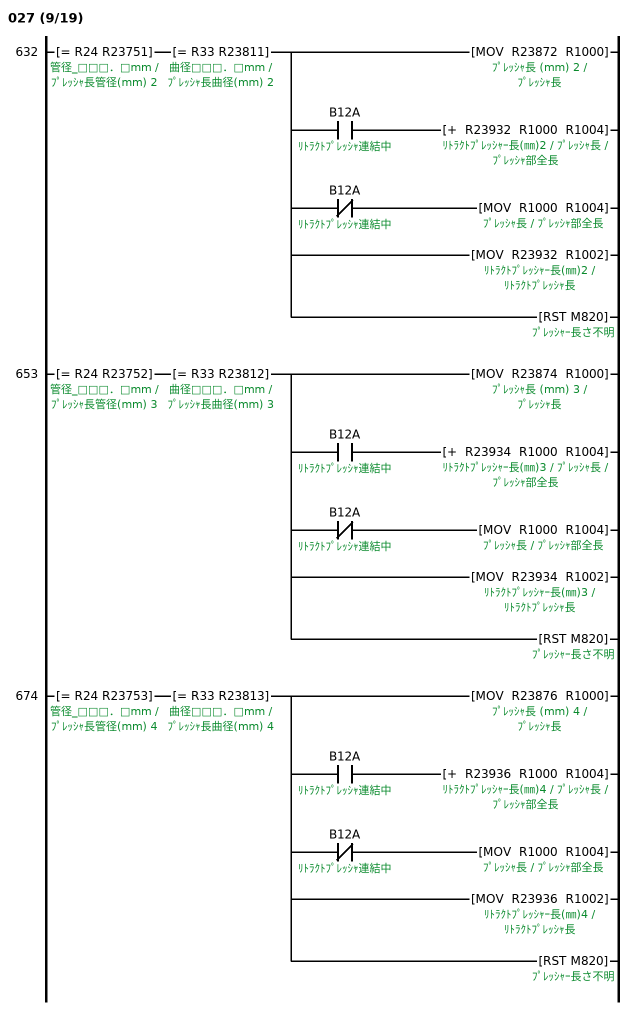
632   LD=     R24 R23751  ; 管径_□□□．□mm / ﾌﾟﾚｯｼｬ長管径(mm) 2
      AND=    R33 R23811  ; 曲径□□□．□mm / ﾌﾟﾚｯｼｬ長曲径(mm) 2
      MOV     R23872 R1000  ; ﾌﾟﾚｯｼｬ長 (mm) 2
      MPS
      AND     B12A  ; ﾘﾄﾗｸﾄﾌﾟﾚｯｼｬ連結中
      +       R23932 R1000 R1004  ; ﾘﾄﾗｸﾄﾌﾟﾚｯｼｬｰ長(㎜)2
      MRD
      ANI     B12A  ; ﾘﾄﾗｸﾄﾌﾟﾚｯｼｬ連結中
      MOV     R1000 R1004
      MPP
      MOV     R23932 R1002
      RST     M820  ; ﾌﾟﾚｯｼｬｰ長さ不明
653   LD=     R24 R23752  ; 管径_□□□．□mm / ﾌﾟﾚｯｼｬ長管径(mm) 3
      AND=    R33 R23812  ; 曲径□□□．□mm / ﾌﾟﾚｯｼｬ長曲径(mm) 3
      MOV     R23874 R1000  ; ﾌﾟﾚｯｼｬ長 (mm) 3
      MPS
      AND     B12A  ; ﾘﾄﾗｸﾄﾌﾟﾚｯｼｬ連結中
      +       R23934 R1000 R1004  ; ﾘﾄﾗｸﾄﾌﾟﾚｯｼｬｰ長(㎜)3
      MRD
      ANI     B12A  ; ﾘﾄﾗｸﾄﾌﾟﾚｯｼｬ連結中
      MOV     R1000 R1004
      MPP
      MOV     R23934 R1002
      RST     M820  ; ﾌﾟﾚｯｼｬｰ長さ不明
674   LD=     R24 R23753  ; 管径_□□□．□mm / ﾌﾟﾚｯｼｬ長管径(mm) 4
      AND=    R33 R23813  ; 曲径□□□．□mm / ﾌﾟﾚｯｼｬ長曲径(mm) 4
      MOV     R23876 R1000  ; ﾌﾟﾚｯｼｬ長 (mm) 4
      MPS
      AND     B12A  ; ﾘﾄﾗｸﾄﾌﾟﾚｯｼｬ連結中
      +       R23936 R1000 R1004  ; ﾘﾄﾗｸﾄﾌﾟﾚｯｼｬｰ長(㎜)4
      MRD
      ANI     B12A  ; ﾘﾄﾗｸﾄﾌﾟﾚｯｼｬ連結中
      MOV     R1000 R1004
      MPP
      MOV     R23936 R1002
      RST     M820  ; ﾌﾟﾚｯｼｬｰ長さ不明
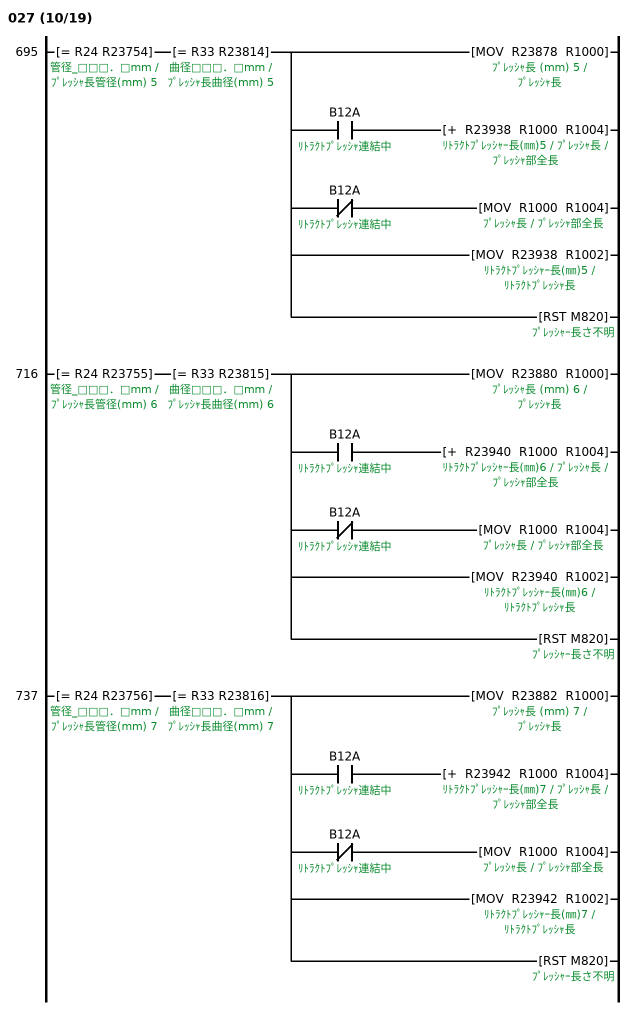
695   LD=     R24 R23754  ; 管径_□□□．□mm / ﾌﾟﾚｯｼｬ長管径(mm) 5
      AND=    R33 R23814  ; 曲径□□□．□mm / ﾌﾟﾚｯｼｬ長曲径(mm) 5
      MOV     R23878 R1000  ; ﾌﾟﾚｯｼｬ長 (mm) 5
      MPS
      AND     B12A  ; ﾘﾄﾗｸﾄﾌﾟﾚｯｼｬ連結中
      +       R23938 R1000 R1004  ; ﾘﾄﾗｸﾄﾌﾟﾚｯｼｬｰ長(㎜)5
      MRD
      ANI     B12A  ; ﾘﾄﾗｸﾄﾌﾟﾚｯｼｬ連結中
      MOV     R1000 R1004
      MPP
      MOV     R23938 R1002
      RST     M820  ; ﾌﾟﾚｯｼｬｰ長さ不明
716   LD=     R24 R23755  ; 管径_□□□．□mm / ﾌﾟﾚｯｼｬ長管径(mm) 6
      AND=    R33 R23815  ; 曲径□□□．□mm / ﾌﾟﾚｯｼｬ長曲径(mm) 6
      MOV     R23880 R1000  ; ﾌﾟﾚｯｼｬ長 (mm) 6
      MPS
      AND     B12A  ; ﾘﾄﾗｸﾄﾌﾟﾚｯｼｬ連結中
      +       R23940 R1000 R1004  ; ﾘﾄﾗｸﾄﾌﾟﾚｯｼｬｰ長(㎜)6
      MRD
      ANI     B12A  ; ﾘﾄﾗｸﾄﾌﾟﾚｯｼｬ連結中
      MOV     R1000 R1004
      MPP
      MOV     R23940 R1002
      RST     M820  ; ﾌﾟﾚｯｼｬｰ長さ不明
737   LD=     R24 R23756  ; 管径_□□□．□mm / ﾌﾟﾚｯｼｬ長管径(mm) 7
      AND=    R33 R23816  ; 曲径□□□．□mm / ﾌﾟﾚｯｼｬ長曲径(mm) 7
      MOV     R23882 R1000  ; ﾌﾟﾚｯｼｬ長 (mm) 7
      MPS
      AND     B12A  ; ﾘﾄﾗｸﾄﾌﾟﾚｯｼｬ連結中
      +       R23942 R1000 R1004  ; ﾘﾄﾗｸﾄﾌﾟﾚｯｼｬｰ長(㎜)7
      MRD
      ANI     B12A  ; ﾘﾄﾗｸﾄﾌﾟﾚｯｼｬ連結中
      MOV     R1000 R1004
      MPP
      MOV     R23942 R1002
      RST     M820  ; ﾌﾟﾚｯｼｬｰ長さ不明
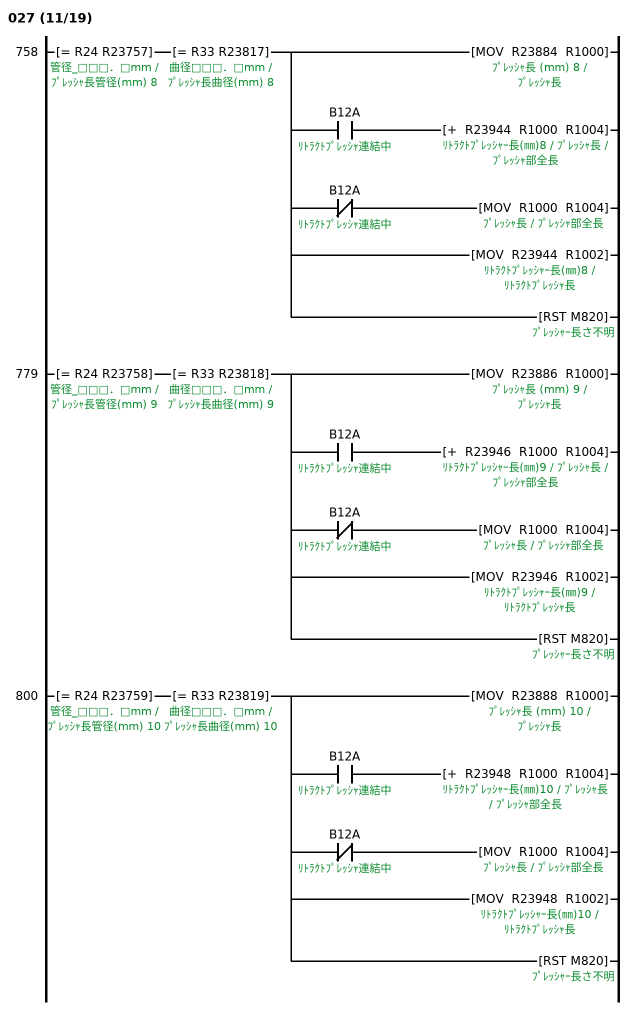
758   LD=     R24 R23757  ; 管径_□□□．□mm / ﾌﾟﾚｯｼｬ長管径(mm) 8
      AND=    R33 R23817  ; 曲径□□□．□mm / ﾌﾟﾚｯｼｬ長曲径(mm) 8
      MOV     R23884 R1000  ; ﾌﾟﾚｯｼｬ長 (mm) 8
      MPS
      AND     B12A  ; ﾘﾄﾗｸﾄﾌﾟﾚｯｼｬ連結中
      +       R23944 R1000 R1004  ; ﾘﾄﾗｸﾄﾌﾟﾚｯｼｬｰ長(㎜)8
      MRD
      ANI     B12A  ; ﾘﾄﾗｸﾄﾌﾟﾚｯｼｬ連結中
      MOV     R1000 R1004
      MPP
      MOV     R23944 R1002
      RST     M820  ; ﾌﾟﾚｯｼｬｰ長さ不明
779   LD=     R24 R23758  ; 管径_□□□．□mm / ﾌﾟﾚｯｼｬ長管径(mm) 9
      AND=    R33 R23818  ; 曲径□□□．□mm / ﾌﾟﾚｯｼｬ長曲径(mm) 9
      MOV     R23886 R1000  ; ﾌﾟﾚｯｼｬ長 (mm) 9
      MPS
      AND     B12A  ; ﾘﾄﾗｸﾄﾌﾟﾚｯｼｬ連結中
      +       R23946 R1000 R1004  ; ﾘﾄﾗｸﾄﾌﾟﾚｯｼｬｰ長(㎜)9
      MRD
      ANI     B12A  ; ﾘﾄﾗｸﾄﾌﾟﾚｯｼｬ連結中
      MOV     R1000 R1004
      MPP
      MOV     R23946 R1002
      RST     M820  ; ﾌﾟﾚｯｼｬｰ長さ不明
800   LD=     R24 R23759  ; 管径_□□□．□mm / ﾌﾟﾚｯｼｬ長管径(mm) 10
      AND=    R33 R23819  ; 曲径□□□．□mm / ﾌﾟﾚｯｼｬ長曲径(mm) 10
      MOV     R23888 R1000  ; ﾌﾟﾚｯｼｬ長 (mm) 10
      MPS
      AND     B12A  ; ﾘﾄﾗｸﾄﾌﾟﾚｯｼｬ連結中
      +       R23948 R1000 R1004  ; ﾘﾄﾗｸﾄﾌﾟﾚｯｼｬｰ長(㎜)10
      MRD
      ANI     B12A  ; ﾘﾄﾗｸﾄﾌﾟﾚｯｼｬ連結中
      MOV     R1000 R1004
      MPP
      MOV     R23948 R1002
      RST     M820  ; ﾌﾟﾚｯｼｬｰ長さ不明
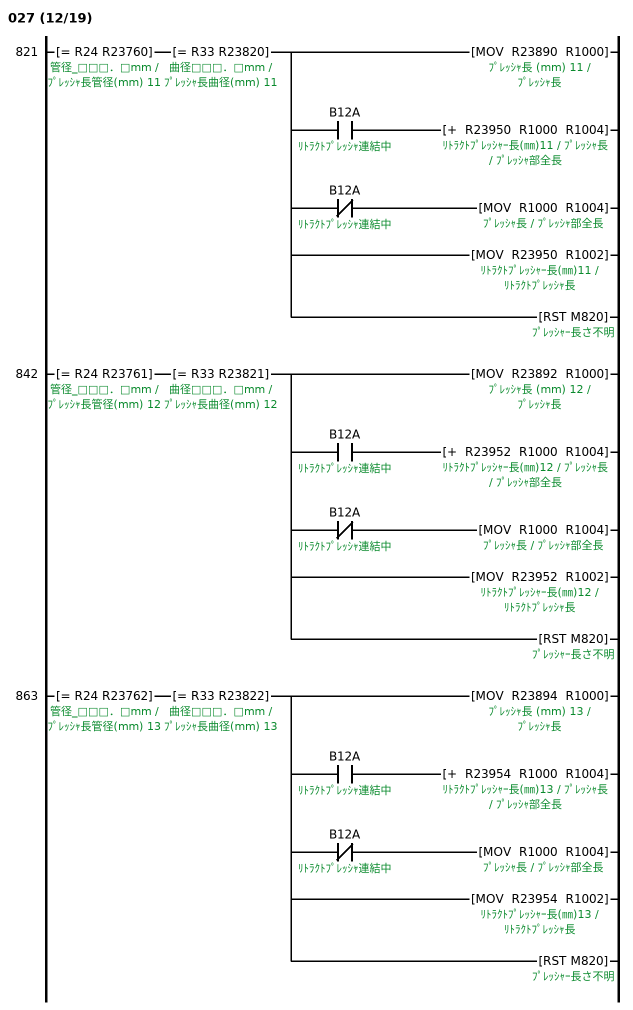
821   LD=     R24 R23760  ; 管径_□□□．□mm / ﾌﾟﾚｯｼｬ長管径(mm) 11
      AND=    R33 R23820  ; 曲径□□□．□mm / ﾌﾟﾚｯｼｬ長曲径(mm) 11
      MOV     R23890 R1000  ; ﾌﾟﾚｯｼｬ長 (mm) 11
      MPS
      AND     B12A  ; ﾘﾄﾗｸﾄﾌﾟﾚｯｼｬ連結中
      +       R23950 R1000 R1004  ; ﾘﾄﾗｸﾄﾌﾟﾚｯｼｬｰ長(㎜)11
      MRD
      ANI     B12A  ; ﾘﾄﾗｸﾄﾌﾟﾚｯｼｬ連結中
      MOV     R1000 R1004
      MPP
      MOV     R23950 R1002
      RST     M820  ; ﾌﾟﾚｯｼｬｰ長さ不明
842   LD=     R24 R23761  ; 管径_□□□．□mm / ﾌﾟﾚｯｼｬ長管径(mm) 12
      AND=    R33 R23821  ; 曲径□□□．□mm / ﾌﾟﾚｯｼｬ長曲径(mm) 12
      MOV     R23892 R1000  ; ﾌﾟﾚｯｼｬ長 (mm) 12
      MPS
      AND     B12A  ; ﾘﾄﾗｸﾄﾌﾟﾚｯｼｬ連結中
      +       R23952 R1000 R1004  ; ﾘﾄﾗｸﾄﾌﾟﾚｯｼｬｰ長(㎜)12
      MRD
      ANI     B12A  ; ﾘﾄﾗｸﾄﾌﾟﾚｯｼｬ連結中
      MOV     R1000 R1004
      MPP
      MOV     R23952 R1002
      RST     M820  ; ﾌﾟﾚｯｼｬｰ長さ不明
863   LD=     R24 R23762  ; 管径_□□□．□mm / ﾌﾟﾚｯｼｬ長管径(mm) 13
      AND=    R33 R23822  ; 曲径□□□．□mm / ﾌﾟﾚｯｼｬ長曲径(mm) 13
      MOV     R23894 R1000  ; ﾌﾟﾚｯｼｬ長 (mm) 13
      MPS
      AND     B12A  ; ﾘﾄﾗｸﾄﾌﾟﾚｯｼｬ連結中
      +       R23954 R1000 R1004  ; ﾘﾄﾗｸﾄﾌﾟﾚｯｼｬｰ長(㎜)13
      MRD
      ANI     B12A  ; ﾘﾄﾗｸﾄﾌﾟﾚｯｼｬ連結中
      MOV     R1000 R1004
      MPP
      MOV     R23954 R1002
      RST     M820  ; ﾌﾟﾚｯｼｬｰ長さ不明
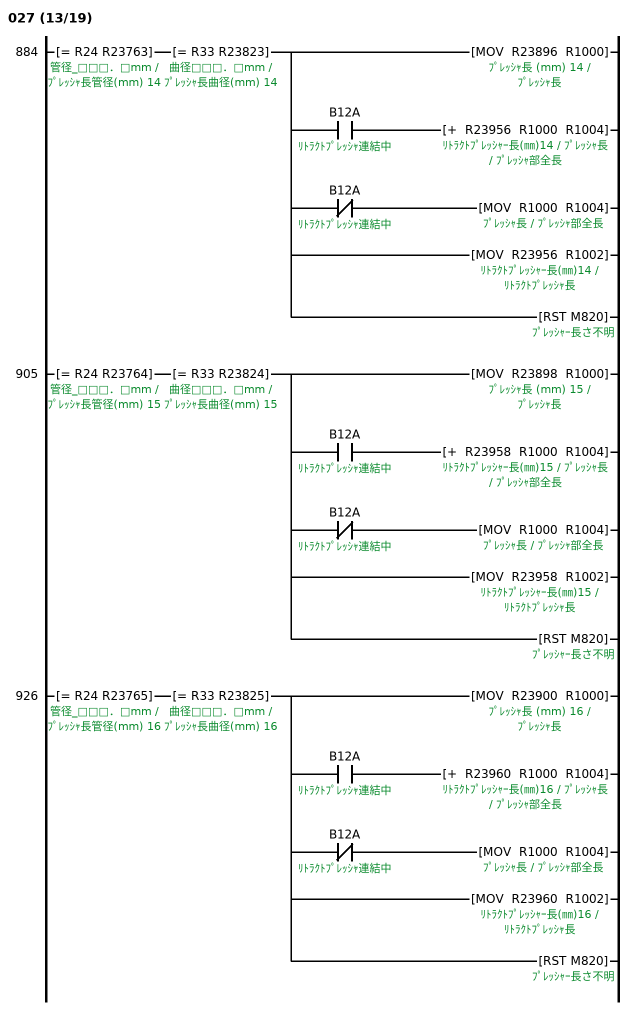
884   LD=     R24 R23763  ; 管径_□□□．□mm / ﾌﾟﾚｯｼｬ長管径(mm) 14
      AND=    R33 R23823  ; 曲径□□□．□mm / ﾌﾟﾚｯｼｬ長曲径(mm) 14
      MOV     R23896 R1000  ; ﾌﾟﾚｯｼｬ長 (mm) 14
      MPS
      AND     B12A  ; ﾘﾄﾗｸﾄﾌﾟﾚｯｼｬ連結中
      +       R23956 R1000 R1004  ; ﾘﾄﾗｸﾄﾌﾟﾚｯｼｬｰ長(㎜)14
      MRD
      ANI     B12A  ; ﾘﾄﾗｸﾄﾌﾟﾚｯｼｬ連結中
      MOV     R1000 R1004
      MPP
      MOV     R23956 R1002
      RST     M820  ; ﾌﾟﾚｯｼｬｰ長さ不明
905   LD=     R24 R23764  ; 管径_□□□．□mm / ﾌﾟﾚｯｼｬ長管径(mm) 15
      AND=    R33 R23824  ; 曲径□□□．□mm / ﾌﾟﾚｯｼｬ長曲径(mm) 15
      MOV     R23898 R1000  ; ﾌﾟﾚｯｼｬ長 (mm) 15
      MPS
      AND     B12A  ; ﾘﾄﾗｸﾄﾌﾟﾚｯｼｬ連結中
      +       R23958 R1000 R1004  ; ﾘﾄﾗｸﾄﾌﾟﾚｯｼｬｰ長(㎜)15
      MRD
      ANI     B12A  ; ﾘﾄﾗｸﾄﾌﾟﾚｯｼｬ連結中
      MOV     R1000 R1004
      MPP
      MOV     R23958 R1002
      RST     M820  ; ﾌﾟﾚｯｼｬｰ長さ不明
926   LD=     R24 R23765  ; 管径_□□□．□mm / ﾌﾟﾚｯｼｬ長管径(mm) 16
      AND=    R33 R23825  ; 曲径□□□．□mm / ﾌﾟﾚｯｼｬ長曲径(mm) 16
      MOV     R23900 R1000  ; ﾌﾟﾚｯｼｬ長 (mm) 16
      MPS
      AND     B12A  ; ﾘﾄﾗｸﾄﾌﾟﾚｯｼｬ連結中
      +       R23960 R1000 R1004  ; ﾘﾄﾗｸﾄﾌﾟﾚｯｼｬｰ長(㎜)16
      MRD
      ANI     B12A  ; ﾘﾄﾗｸﾄﾌﾟﾚｯｼｬ連結中
      MOV     R1000 R1004
      MPP
      MOV     R23960 R1002
      RST     M820  ; ﾌﾟﾚｯｼｬｰ長さ不明
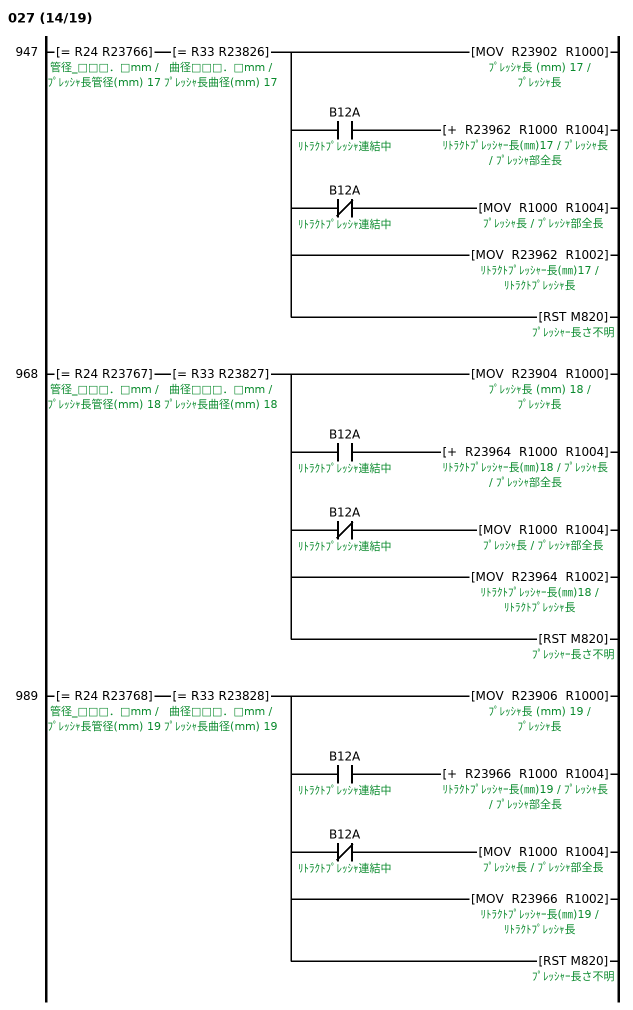
947   LD=     R24 R23766  ; 管径_□□□．□mm / ﾌﾟﾚｯｼｬ長管径(mm) 17
      AND=    R33 R23826  ; 曲径□□□．□mm / ﾌﾟﾚｯｼｬ長曲径(mm) 17
      MOV     R23902 R1000  ; ﾌﾟﾚｯｼｬ長 (mm) 17
      MPS
      AND     B12A  ; ﾘﾄﾗｸﾄﾌﾟﾚｯｼｬ連結中
      +       R23962 R1000 R1004  ; ﾘﾄﾗｸﾄﾌﾟﾚｯｼｬｰ長(㎜)17
      MRD
      ANI     B12A  ; ﾘﾄﾗｸﾄﾌﾟﾚｯｼｬ連結中
      MOV     R1000 R1004
      MPP
      MOV     R23962 R1002
      RST     M820  ; ﾌﾟﾚｯｼｬｰ長さ不明
968   LD=     R24 R23767  ; 管径_□□□．□mm / ﾌﾟﾚｯｼｬ長管径(mm) 18
      AND=    R33 R23827  ; 曲径□□□．□mm / ﾌﾟﾚｯｼｬ長曲径(mm) 18
      MOV     R23904 R1000  ; ﾌﾟﾚｯｼｬ長 (mm) 18
      MPS
      AND     B12A  ; ﾘﾄﾗｸﾄﾌﾟﾚｯｼｬ連結中
      +       R23964 R1000 R1004  ; ﾘﾄﾗｸﾄﾌﾟﾚｯｼｬｰ長(㎜)18
      MRD
      ANI     B12A  ; ﾘﾄﾗｸﾄﾌﾟﾚｯｼｬ連結中
      MOV     R1000 R1004
      MPP
      MOV     R23964 R1002
      RST     M820  ; ﾌﾟﾚｯｼｬｰ長さ不明
989   LD=     R24 R23768  ; 管径_□□□．□mm / ﾌﾟﾚｯｼｬ長管径(mm) 19
      AND=    R33 R23828  ; 曲径□□□．□mm / ﾌﾟﾚｯｼｬ長曲径(mm) 19
      MOV     R23906 R1000  ; ﾌﾟﾚｯｼｬ長 (mm) 19
      MPS
      AND     B12A  ; ﾘﾄﾗｸﾄﾌﾟﾚｯｼｬ連結中
      +       R23966 R1000 R1004  ; ﾘﾄﾗｸﾄﾌﾟﾚｯｼｬｰ長(㎜)19
      MRD
      ANI     B12A  ; ﾘﾄﾗｸﾄﾌﾟﾚｯｼｬ連結中
      MOV     R1000 R1004
      MPP
      MOV     R23966 R1002
      RST     M820  ; ﾌﾟﾚｯｼｬｰ長さ不明
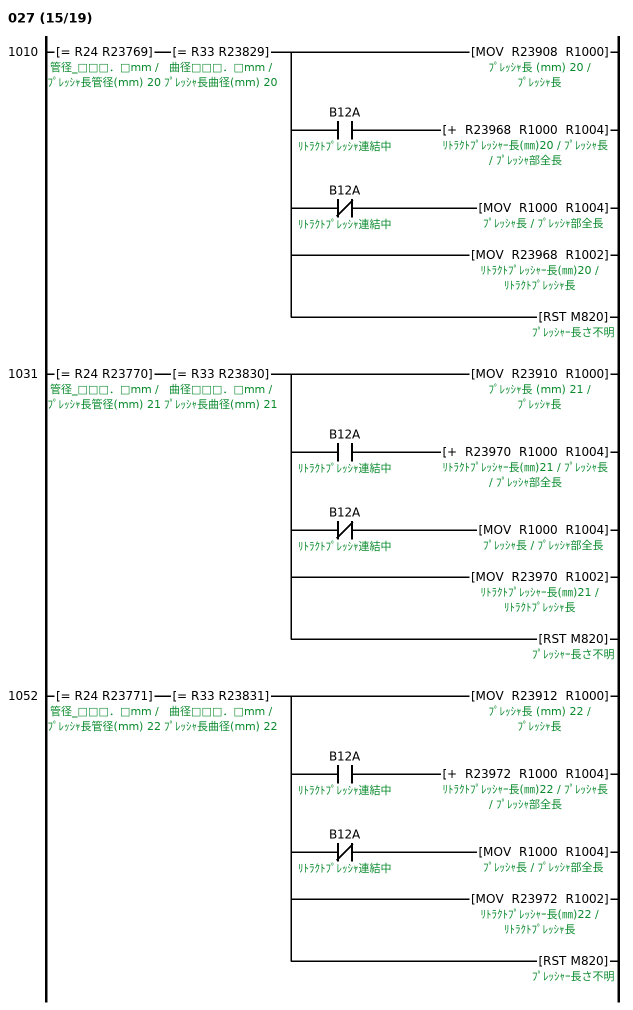
1010  LD=     R24 R23769  ; 管径_□□□．□mm / ﾌﾟﾚｯｼｬ長管径(mm) 20
      AND=    R33 R23829  ; 曲径□□□．□mm / ﾌﾟﾚｯｼｬ長曲径(mm) 20
      MOV     R23908 R1000  ; ﾌﾟﾚｯｼｬ長 (mm) 20
      MPS
      AND     B12A  ; ﾘﾄﾗｸﾄﾌﾟﾚｯｼｬ連結中
      +       R23968 R1000 R1004  ; ﾘﾄﾗｸﾄﾌﾟﾚｯｼｬｰ長(㎜)20
      MRD
      ANI     B12A  ; ﾘﾄﾗｸﾄﾌﾟﾚｯｼｬ連結中
      MOV     R1000 R1004
      MPP
      MOV     R23968 R1002
      RST     M820  ; ﾌﾟﾚｯｼｬｰ長さ不明
1031  LD=     R24 R23770  ; 管径_□□□．□mm / ﾌﾟﾚｯｼｬ長管径(mm) 21
      AND=    R33 R23830  ; 曲径□□□．□mm / ﾌﾟﾚｯｼｬ長曲径(mm) 21
      MOV     R23910 R1000  ; ﾌﾟﾚｯｼｬ長 (mm) 21
      MPS
      AND     B12A  ; ﾘﾄﾗｸﾄﾌﾟﾚｯｼｬ連結中
      +       R23970 R1000 R1004  ; ﾘﾄﾗｸﾄﾌﾟﾚｯｼｬｰ長(㎜)21
      MRD
      ANI     B12A  ; ﾘﾄﾗｸﾄﾌﾟﾚｯｼｬ連結中
      MOV     R1000 R1004
      MPP
      MOV     R23970 R1002
      RST     M820  ; ﾌﾟﾚｯｼｬｰ長さ不明
1052  LD=     R24 R23771  ; 管径_□□□．□mm / ﾌﾟﾚｯｼｬ長管径(mm) 22
      AND=    R33 R23831  ; 曲径□□□．□mm / ﾌﾟﾚｯｼｬ長曲径(mm) 22
      MOV     R23912 R1000  ; ﾌﾟﾚｯｼｬ長 (mm) 22
      MPS
      AND     B12A  ; ﾘﾄﾗｸﾄﾌﾟﾚｯｼｬ連結中
      +       R23972 R1000 R1004  ; ﾘﾄﾗｸﾄﾌﾟﾚｯｼｬｰ長(㎜)22
      MRD
      ANI     B12A  ; ﾘﾄﾗｸﾄﾌﾟﾚｯｼｬ連結中
      MOV     R1000 R1004
      MPP
      MOV     R23972 R1002
      RST     M820  ; ﾌﾟﾚｯｼｬｰ長さ不明
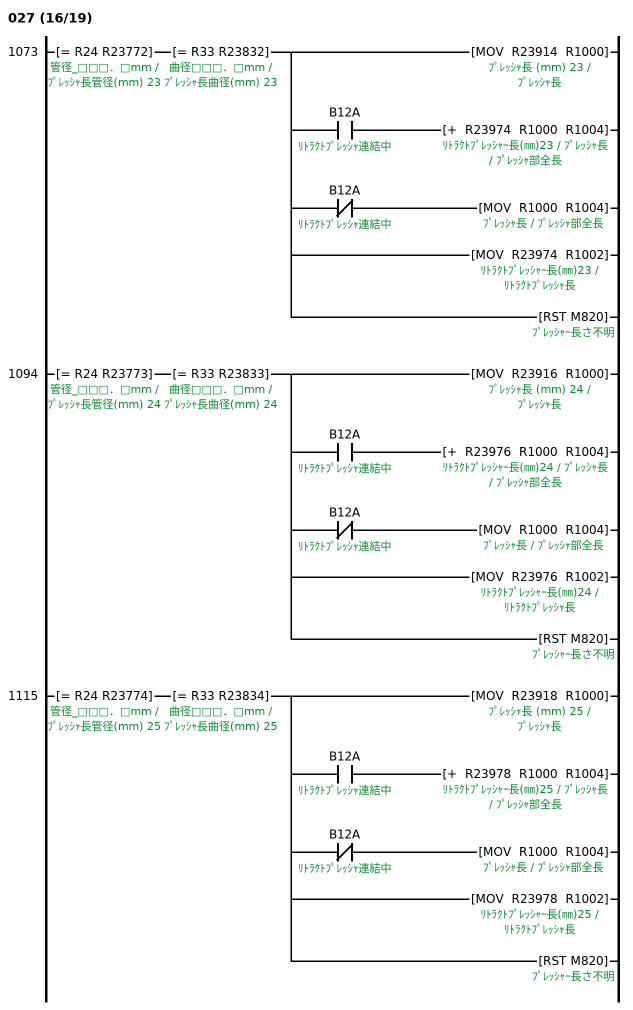
1073  LD=     R24 R23772  ; 管径_□□□．□mm / ﾌﾟﾚｯｼｬ長管径(mm) 23
      AND=    R33 R23832  ; 曲径□□□．□mm / ﾌﾟﾚｯｼｬ長曲径(mm) 23
      MOV     R23914 R1000  ; ﾌﾟﾚｯｼｬ長 (mm) 23
      MPS
      AND     B12A  ; ﾘﾄﾗｸﾄﾌﾟﾚｯｼｬ連結中
      +       R23974 R1000 R1004  ; ﾘﾄﾗｸﾄﾌﾟﾚｯｼｬｰ長(㎜)23
      MRD
      ANI     B12A  ; ﾘﾄﾗｸﾄﾌﾟﾚｯｼｬ連結中
      MOV     R1000 R1004
      MPP
      MOV     R23974 R1002
      RST     M820  ; ﾌﾟﾚｯｼｬｰ長さ不明
1094  LD=     R24 R23773  ; 管径_□□□．□mm / ﾌﾟﾚｯｼｬ長管径(mm) 24
      AND=    R33 R23833  ; 曲径□□□．□mm / ﾌﾟﾚｯｼｬ長曲径(mm) 24
      MOV     R23916 R1000  ; ﾌﾟﾚｯｼｬ長 (mm) 24
      MPS
      AND     B12A  ; ﾘﾄﾗｸﾄﾌﾟﾚｯｼｬ連結中
      +       R23976 R1000 R1004  ; ﾘﾄﾗｸﾄﾌﾟﾚｯｼｬｰ長(㎜)24
      MRD
      ANI     B12A  ; ﾘﾄﾗｸﾄﾌﾟﾚｯｼｬ連結中
      MOV     R1000 R1004
      MPP
      MOV     R23976 R1002
      RST     M820  ; ﾌﾟﾚｯｼｬｰ長さ不明
1115  LD=     R24 R23774  ; 管径_□□□．□mm / ﾌﾟﾚｯｼｬ長管径(mm) 25
      AND=    R33 R23834  ; 曲径□□□．□mm / ﾌﾟﾚｯｼｬ長曲径(mm) 25
      MOV     R23918 R1000  ; ﾌﾟﾚｯｼｬ長 (mm) 25
      MPS
      AND     B12A  ; ﾘﾄﾗｸﾄﾌﾟﾚｯｼｬ連結中
      +       R23978 R1000 R1004  ; ﾘﾄﾗｸﾄﾌﾟﾚｯｼｬｰ長(㎜)25
      MRD
      ANI     B12A  ; ﾘﾄﾗｸﾄﾌﾟﾚｯｼｬ連結中
      MOV     R1000 R1004
      MPP
      MOV     R23978 R1002
      RST     M820  ; ﾌﾟﾚｯｼｬｰ長さ不明
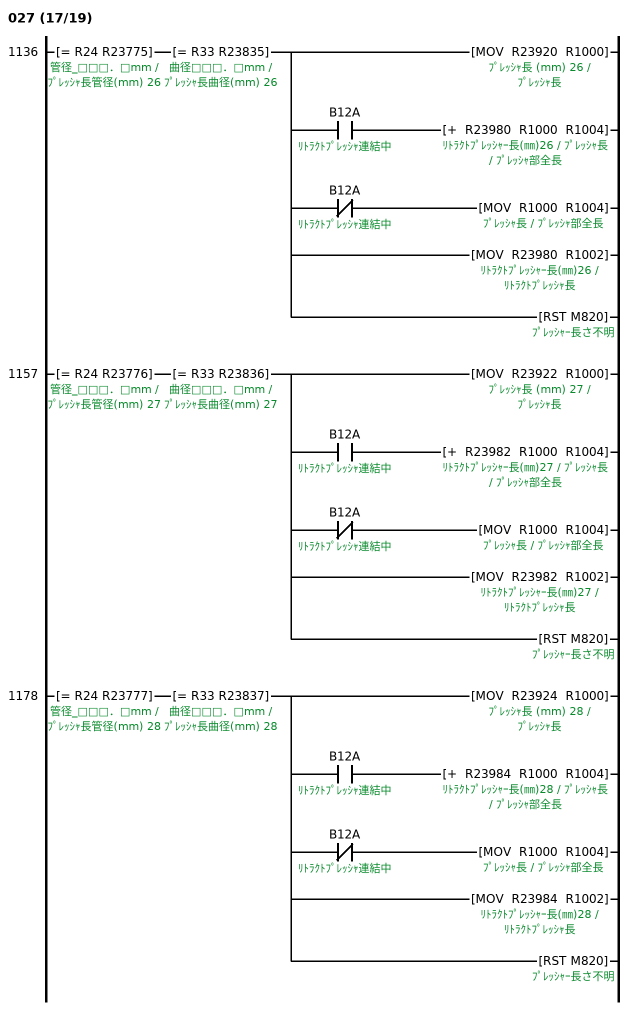
1136  LD=     R24 R23775  ; 管径_□□□．□mm / ﾌﾟﾚｯｼｬ長管径(mm) 26
      AND=    R33 R23835  ; 曲径□□□．□mm / ﾌﾟﾚｯｼｬ長曲径(mm) 26
      MOV     R23920 R1000  ; ﾌﾟﾚｯｼｬ長 (mm) 26
      MPS
      AND     B12A  ; ﾘﾄﾗｸﾄﾌﾟﾚｯｼｬ連結中
      +       R23980 R1000 R1004  ; ﾘﾄﾗｸﾄﾌﾟﾚｯｼｬｰ長(㎜)26
      MRD
      ANI     B12A  ; ﾘﾄﾗｸﾄﾌﾟﾚｯｼｬ連結中
      MOV     R1000 R1004
      MPP
      MOV     R23980 R1002
      RST     M820  ; ﾌﾟﾚｯｼｬｰ長さ不明
1157  LD=     R24 R23776  ; 管径_□□□．□mm / ﾌﾟﾚｯｼｬ長管径(mm) 27
      AND=    R33 R23836  ; 曲径□□□．□mm / ﾌﾟﾚｯｼｬ長曲径(mm) 27
      MOV     R23922 R1000  ; ﾌﾟﾚｯｼｬ長 (mm) 27
      MPS
      AND     B12A  ; ﾘﾄﾗｸﾄﾌﾟﾚｯｼｬ連結中
      +       R23982 R1000 R1004  ; ﾘﾄﾗｸﾄﾌﾟﾚｯｼｬｰ長(㎜)27
      MRD
      ANI     B12A  ; ﾘﾄﾗｸﾄﾌﾟﾚｯｼｬ連結中
      MOV     R1000 R1004
      MPP
      MOV     R23982 R1002
      RST     M820  ; ﾌﾟﾚｯｼｬｰ長さ不明
1178  LD=     R24 R23777  ; 管径_□□□．□mm / ﾌﾟﾚｯｼｬ長管径(mm) 28
      AND=    R33 R23837  ; 曲径□□□．□mm / ﾌﾟﾚｯｼｬ長曲径(mm) 28
      MOV     R23924 R1000  ; ﾌﾟﾚｯｼｬ長 (mm) 28
      MPS
      AND     B12A  ; ﾘﾄﾗｸﾄﾌﾟﾚｯｼｬ連結中
      +       R23984 R1000 R1004  ; ﾘﾄﾗｸﾄﾌﾟﾚｯｼｬｰ長(㎜)28
      MRD
      ANI     B12A  ; ﾘﾄﾗｸﾄﾌﾟﾚｯｼｬ連結中
      MOV     R1000 R1004
      MPP
      MOV     R23984 R1002
      RST     M820  ; ﾌﾟﾚｯｼｬｰ長さ不明
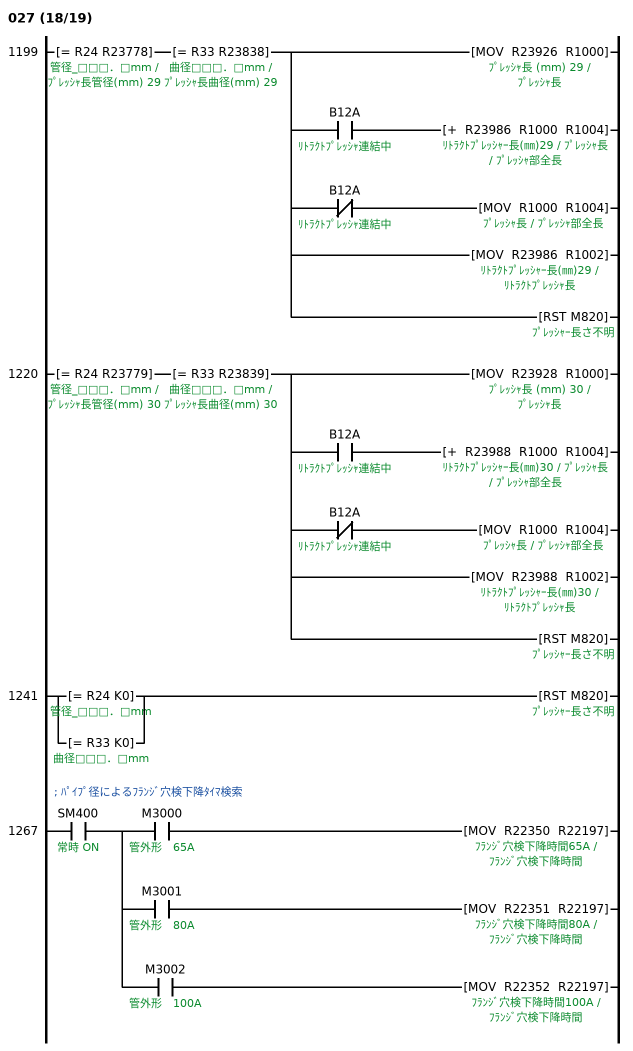
1199  LD=     R24 R23778  ; 管径_□□□．□mm / ﾌﾟﾚｯｼｬ長管径(mm) 29
      AND=    R33 R23838  ; 曲径□□□．□mm / ﾌﾟﾚｯｼｬ長曲径(mm) 29
      MOV     R23926 R1000  ; ﾌﾟﾚｯｼｬ長 (mm) 29
      MPS
      AND     B12A  ; ﾘﾄﾗｸﾄﾌﾟﾚｯｼｬ連結中
      +       R23986 R1000 R1004  ; ﾘﾄﾗｸﾄﾌﾟﾚｯｼｬｰ長(㎜)29
      MRD
      ANI     B12A  ; ﾘﾄﾗｸﾄﾌﾟﾚｯｼｬ連結中
      MOV     R1000 R1004
      MPP
      MOV     R23986 R1002
      RST     M820  ; ﾌﾟﾚｯｼｬｰ長さ不明
1220  LD=     R24 R23779  ; 管径_□□□．□mm / ﾌﾟﾚｯｼｬ長管径(mm) 30
      AND=    R33 R23839  ; 曲径□□□．□mm / ﾌﾟﾚｯｼｬ長曲径(mm) 30
      MOV     R23928 R1000  ; ﾌﾟﾚｯｼｬ長 (mm) 30
      MPS
      AND     B12A  ; ﾘﾄﾗｸﾄﾌﾟﾚｯｼｬ連結中
      +       R23988 R1000 R1004  ; ﾘﾄﾗｸﾄﾌﾟﾚｯｼｬｰ長(㎜)30
      MRD
      ANI     B12A  ; ﾘﾄﾗｸﾄﾌﾟﾚｯｼｬ連結中
      MOV     R1000 R1004
      MPP
      MOV     R23988 R1002
      RST     M820  ; ﾌﾟﾚｯｼｬｰ長さ不明
1241  LD=     R24 K0  ; 管径_□□□．□mm
      OR=     R33 K0  ; 曲径□□□．□mm
      RST     M820  ; ﾌﾟﾚｯｼｬｰ長さ不明
; ﾊﾟｲﾌﾟ径によるﾌﾗﾝｼﾞ穴検下降ﾀｲﾏ検索
1267  LD      SM400  ; 常時 ON
      MPS
      AND     M3000  ; 管外形　65A
      MOV     R22350 R22197  ; ﾌﾗﾝｼﾞ穴検下降時間65A / ﾌﾗﾝｼﾞ穴検下降時間
      MRD
      AND     M3001  ; 管外形　80A
      MOV     R22351 R22197  ; ﾌﾗﾝｼﾞ穴検下降時間80A
      MPP
      AND     M3002  ; 管外形　100A
      MOV     R22352 R22197  ; ﾌﾗﾝｼﾞ穴検下降時間100A
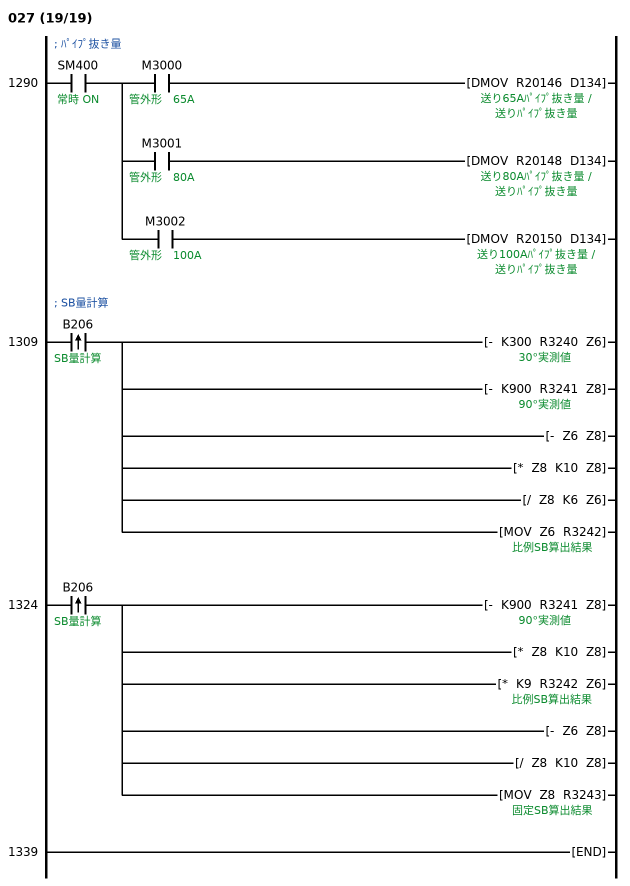
; 
; ﾊﾟｲﾌﾟ抜き量
1290  LD      SM400  ; 常時 ON
      MPS
      AND     M3000  ; 管外形　65A
      DMOV    R20146 D134  ; 送り65Aﾊﾟｲﾌﾟ抜き量 / 送りﾊﾟｲﾌﾟ抜き量
      MRD
      AND     M3001  ; 管外形　80A
      DMOV    R20148 D134  ; 送り80Aﾊﾟｲﾌﾟ抜き量
      MPP
      AND     M3002  ; 管外形　100A
      DMOV    R20150 D134  ; 送り100Aﾊﾟｲﾌﾟ抜き量
; SB量計算
1309  LDP     B206  ; SB量計算
      -       K300 R3240 Z6  ; 30°実測値
      -       K900 R3241 Z8  ; 90°実測値
      -       Z6 Z8
      *       Z8 K10 Z8
      /       Z8 K6 Z6
      MOV     Z6 R3242  ; 比例SB算出結果
1324  LDP     B206  ; SB量計算
      -       K900 R3241 Z8
      *       Z8 K10 Z8
      *       K9 R3242 Z6
      -       Z6 Z8
      /       Z8 K10 Z8
      MOV     Z8 R3243  ; 固定SB算出結果
1339  END
END_PROGRAM

PROGRAM 028  // ﾃﾞｰﾀ変換
; 
      P2800
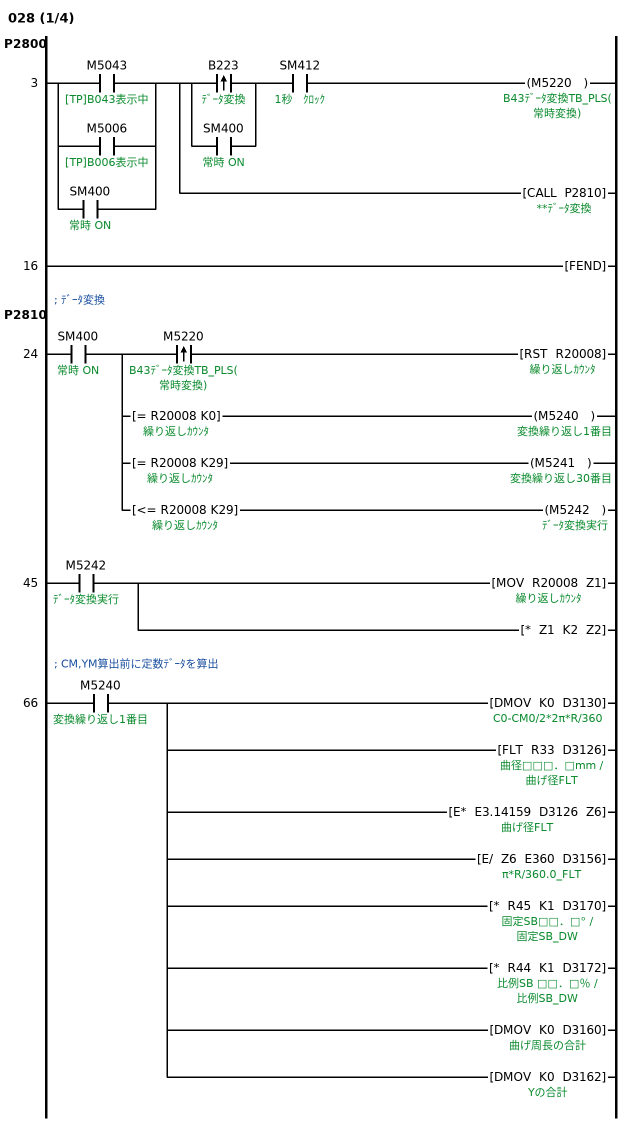
3     LD      M5043  ; [TP]B043表示中
      OR      M5006  ; [TP]B006表示中
      OR      SM400  ; 常時 ON
      MPS
      LDP     B223  ; ﾃﾞｰﾀ変換
      OR      SM400  ; 常時 ON
      ANB
      AND     SM412  ; 1秒   ｸﾛｯｸ
      OUT     M5220  ; B43ﾃﾞｰﾀ変換TB_PLS(常時変換)
      MPP
      CALL    P2810  ; **ﾃﾞｰﾀ変換
16    FEND
; ﾃﾞｰﾀ変換
      P2810
24    LD      SM400  ; 常時 ON
      MPS
      ANDP    M5220  ; B43ﾃﾞｰﾀ変換TB_PLS(常時変換)
      RST     R20008  ; 繰り返しｶｳﾝﾀ
      MRD
      AND=    R20008 K0  ; 繰り返しｶｳﾝﾀ
      OUT     M5240  ; 変換繰り返し1番目
      MRD
      AND=    R20008 K29  ; 繰り返しｶｳﾝﾀ
      OUT     M5241  ; 変換繰り返し30番目
      MPP
      AND<=   R20008 K29  ; 繰り返しｶｳﾝﾀ
      OUT     M5242  ; ﾃﾞｰﾀ変換実行
45    LD      M5242  ; ﾃﾞｰﾀ変換実行
      MOV     R20008 Z1
      *       Z1 K2 Z2
; CM,YM算出前に定数ﾃﾞｰﾀを算出
66    LD      M5240  ; 変換繰り返し1番目
      DMOV    K0 D3130  ; C0-CM0/2*2π*R/360
      FLT     R33 D3126  ; 曲径□□□．□mm / 曲げ径FLT
      E*      E3.14159 D3126 Z6
      E/      Z6 E360 D3156  ; π*R/360.0_FLT
      *       R45 K1 D3170  ; 固定SB□□．□° / 固定SB_DW
      *       R44 K1 D3172  ; 比例SB □□．□％ / 比例SB_DW
      DMOV    K0 D3160  ; 曲げ周長の合計
      DMOV    K0 D3162  ; Yの合計
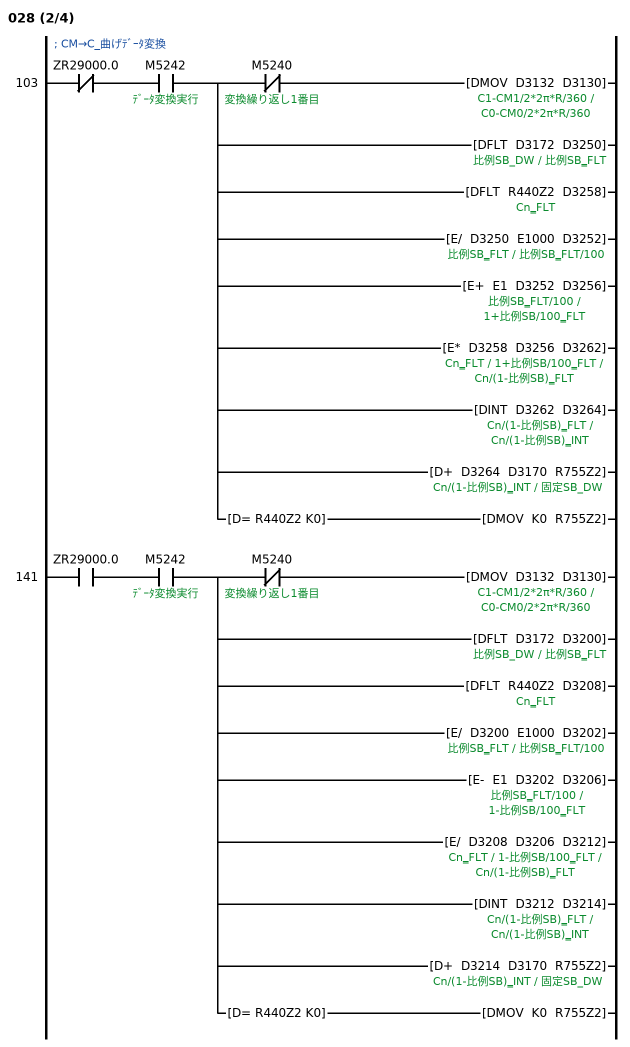
; CM→C_曲げﾃﾞｰﾀ変換
103   LDI     ZR29000.0
      AND     M5242  ; ﾃﾞｰﾀ変換実行
      MPS
      ANI     M5240  ; 変換繰り返し1番目
      DMOV    D3132 D3130  ; C1-CM1/2*2π*R/360
      MPP
      DFLT    D3172 D3250  ; 比例SB‗FLT
      DFLT    R440Z2 D3258  ; Cn‗FLT
      E/      D3250 E1000 D3252  ; 比例SB‗FLT/100
      E+      E1 D3252 D3256  ; 1+比例SB/100‗FLT
      E*      D3258 D3256 D3262  ; Cn/(1-比例SB)‗FLT
      DINT    D3262 D3264  ; Cn/(1-比例SB)‗INT
      D+      D3264 D3170 R755Z2
      ANDD=   R440Z2 K0
      DMOV    K0 R755Z2
141   LD      ZR29000.0
      AND     M5242  ; ﾃﾞｰﾀ変換実行
      MPS
      ANI     M5240  ; 変換繰り返し1番目
      DMOV    D3132 D3130
      MPP
      DFLT    D3172 D3200  ; 比例SB‗FLT
      DFLT    R440Z2 D3208  ; Cn‗FLT
      E/      D3200 E1000 D3202  ; 比例SB‗FLT/100
      E-      E1 D3202 D3206  ; 1-比例SB/100‗FLT
      E/      D3208 D3206 D3212  ; Cn/(1-比例SB)‗FLT
      DINT    D3212 D3214  ; Cn/(1-比例SB)‗INT
      D+      D3214 D3170 R755Z2
      ANDD=   R440Z2 K0
      DMOV    K0 R755Z2
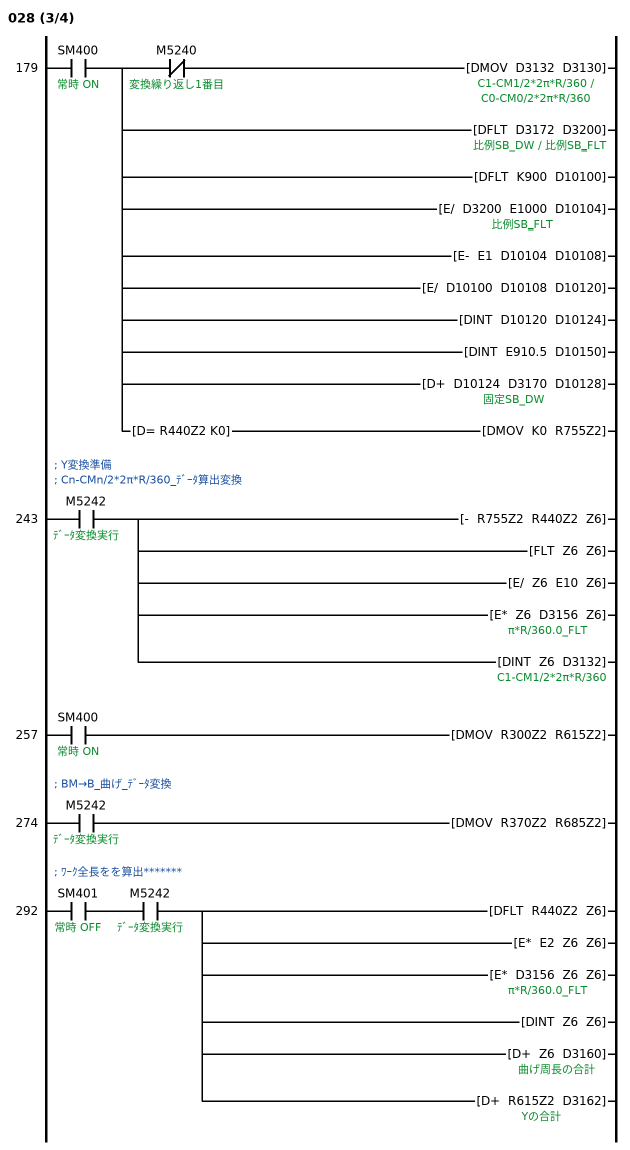
179   LD      SM400  ; 常時 ON
      MPS
      ANI     M5240  ; 変換繰り返し1番目
      DMOV    D3132 D3130
      MPP
      DFLT    D3172 D3200
      DFLT    K900 D10100
      E/      D3200 E1000 D10104
      E-      E1 D10104 D10108
      E/      D10100 D10108 D10120
      DINT    D10120 D10124
      DINT    E910.5 D10150
      D+      D10124 D3170 D10128
      ANDD=   R440Z2 K0
      DMOV    K0 R755Z2
; Y変換準備
; Cn-CMn/2*2π*R/360_ﾃﾞｰﾀ算出変換
243   LD      M5242  ; ﾃﾞｰﾀ変換実行
      -       R755Z2 R440Z2 Z6
      FLT     Z6 Z6
      E/      Z6 E10 Z6
      E*      Z6 D3156 Z6
      DINT    Z6 D3132
257   LD      SM400  ; 常時 ON
      DMOV    R300Z2 R615Z2
; BM→B_曲げ_ﾃﾞｰﾀ変換
274   LD      M5242  ; ﾃﾞｰﾀ変換実行
      DMOV    R370Z2 R685Z2
; ﾜｰｸ全長をを算出*******
292   LD      SM401  ; 常時 OFF
      AND     M5242  ; ﾃﾞｰﾀ変換実行
      DFLT    R440Z2 Z6
      E*      E2 Z6 Z6
      E*      D3156 Z6 Z6
      DINT    Z6 Z6
      D+      Z6 D3160
      D+      R615Z2 D3162
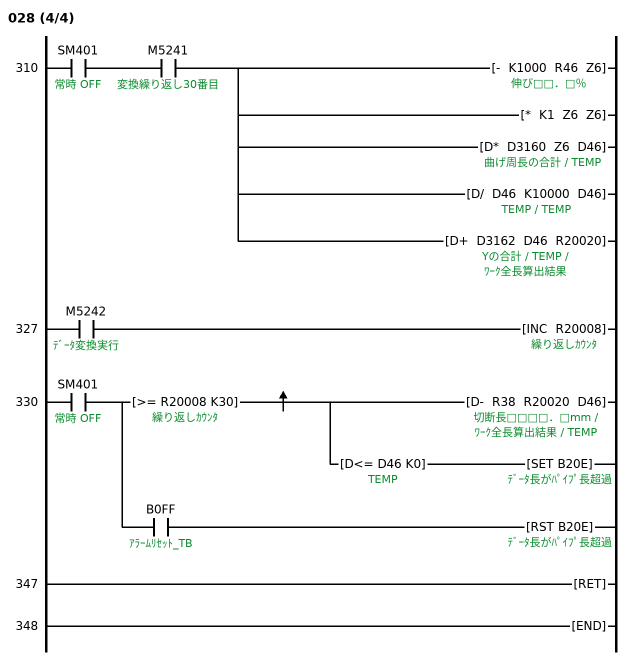
310   LD      SM401  ; 常時 OFF
      AND     M5241  ; 変換繰り返し30番目
      -       K1000 R46 Z6  ; 伸び□□．□％
      *       K1 Z6 Z6
      D*      D3160 Z6 D46  ; TEMP
      D/      D46 K10000 D46
      D+      D3162 D46 R20020  ; ﾜｰｸ全長算出結果
327   LD      M5242  ; ﾃﾞｰﾀ変換実行
      INC     R20008
330   LD      SM401  ; 常時 OFF
      MPS
      AND>=   R20008 K30  ; 繰り返しｶｳﾝﾀ
      MEP
      D-      R38 R20020 D46  ; 切断長□□□□．□mm
      ANDD<=  D46 K0  ; TEMP
      SET     B20E  ; ﾃﾞｰﾀ長がﾊﾟｲﾌﾟ長超過
      MPP
      AND     B0FF  ; ｱﾗｰﾑﾘｾｯﾄ_TB
      RST     B20E  ; ﾃﾞｰﾀ長がﾊﾟｲﾌﾟ長超過
347   RET
348   END
END_PROGRAM

PROGRAM 029  // 出力
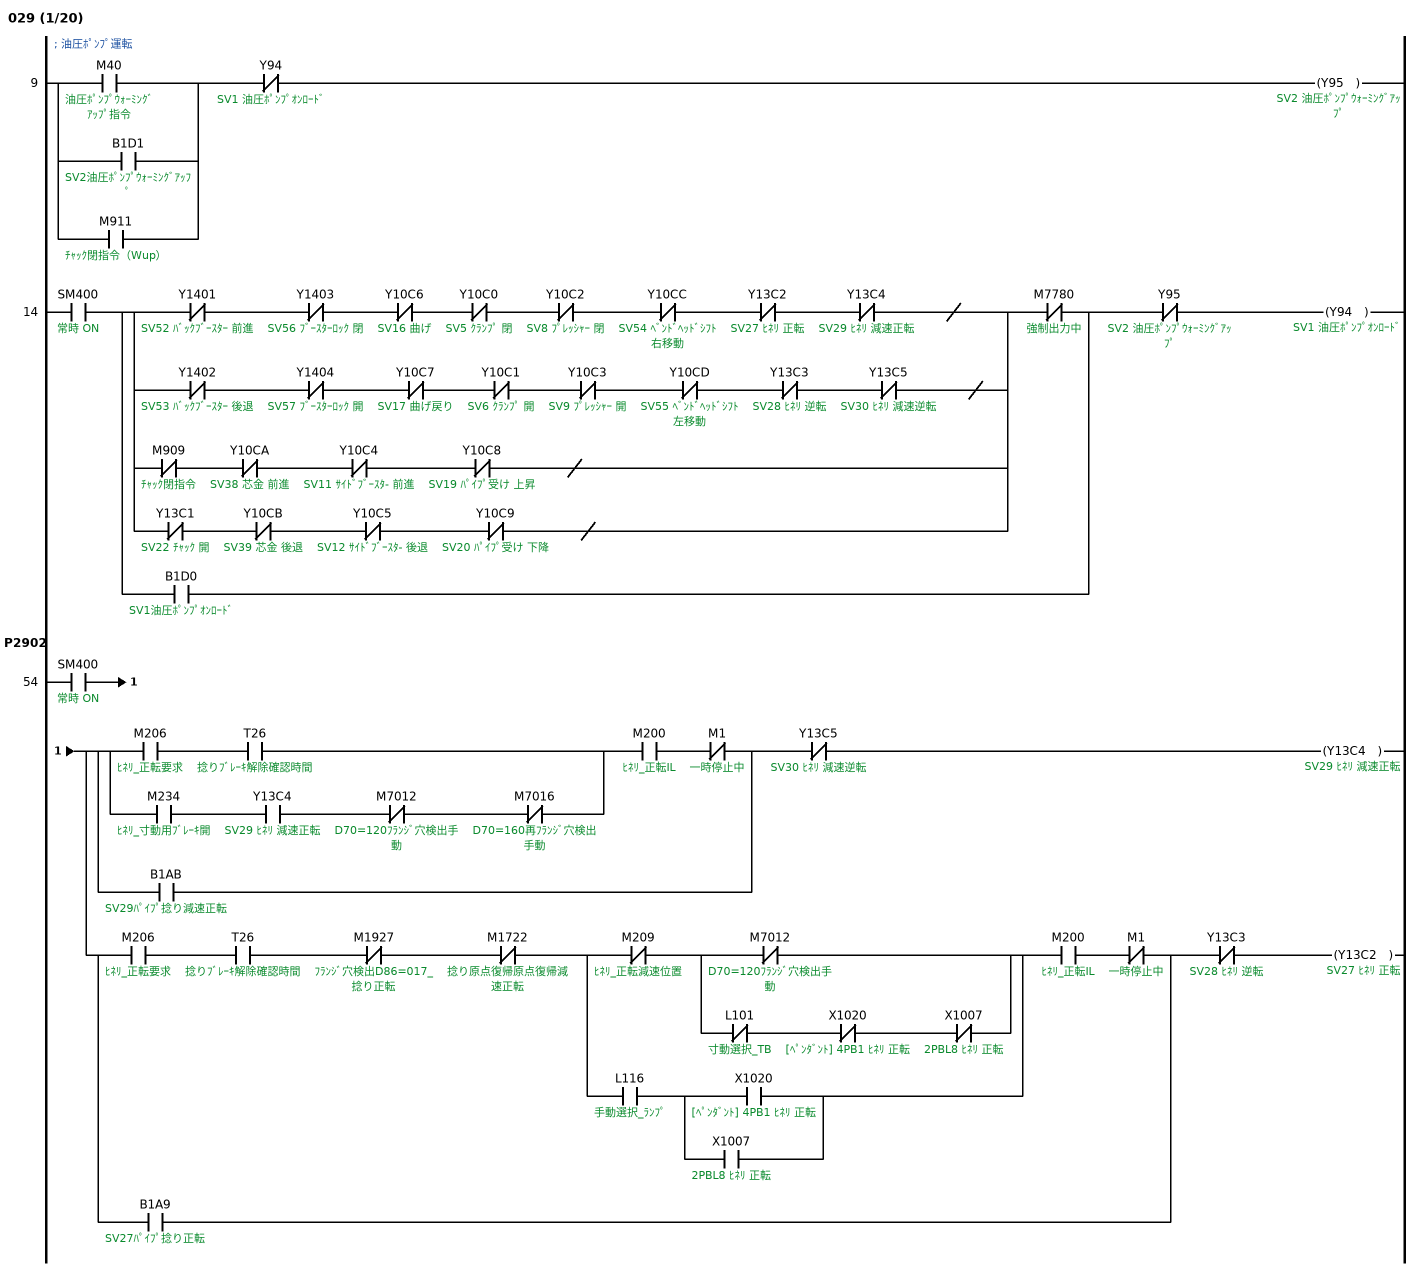
; 油圧ﾎﾟﾝﾌﾟ運転
9     LD      M40  ; 油圧ﾎﾟﾝﾌﾟｳｫｰﾐﾝｸﾞ ｱｯﾌﾟ指令
      OR      B1D1  ; SV2油圧ﾎﾟﾝﾌﾟｳｫｰﾐﾝｸﾞｱｯﾌﾟ
      OR      M911  ; ﾁｬｯｸ閉指令（Wup）
      ANI     Y94  ; SV1 油圧ﾎﾟﾝﾌﾟｵﾝﾛｰﾄﾞ
      OUT     Y95  ; SV2 油圧ﾎﾟﾝﾌﾟｳｫｰﾐﾝｸﾞｱｯﾌﾟ
14    LD      SM400  ; 常時 ON
      LDI     Y1401  ; SV52 ﾊﾞｯｸﾌﾞｰｽﾀｰ 前進
      ANI     Y1403  ; SV56 ﾌﾞｰｽﾀｰﾛｯｸ 閉
      ANI     Y10C6  ; SV16 曲げ
      ANI     Y10C0  ; SV5 ｸﾗﾝﾌﾟ 閉
      ANI     Y10C2  ; SV8 ﾌﾟﾚｯｼｬｰ 閉
      ANI     Y10CC  ; SV54 ﾍﾞﾝﾄﾞﾍｯﾄﾞｼﾌﾄ 右移動
      ANI     Y13C2  ; SV27 ﾋﾈﾘ 正転
      ANI     Y13C4  ; SV29 ﾋﾈﾘ 減速正転
      INV
      LDI     Y1402  ; SV53 ﾊﾞｯｸﾌﾞｰｽﾀｰ 後退
      ANI     Y1404  ; SV57 ﾌﾞｰｽﾀｰﾛｯｸ 開
      ANI     Y10C7  ; SV17 曲げ戻り
      ANI     Y10C1  ; SV6 ｸﾗﾝﾌﾟ 開
      ANI     Y10C3  ; SV9 ﾌﾟﾚｯｼｬｰ 開
      ANI     Y10CD  ; SV55 ﾍﾞﾝﾄﾞﾍｯﾄﾞｼﾌﾄ 左移動
      ANI     Y13C3  ; SV28 ﾋﾈﾘ 逆転
      ANI     Y13C5  ; SV30 ﾋﾈﾘ 減速逆転
      INV
      ORB
      LDI     M909  ; ﾁｬｯｸ閉指令
      ANI     Y10CA  ; SV38 芯金 前進
      ANI     Y10C4  ; SV11 ｻｲﾄﾞﾌﾞｰｽﾀ- 前進
      ANI     Y10C8  ; SV19 ﾊﾟｲﾌﾟ受け 上昇
      INV
      ORB
      LDI     Y13C1  ; SV22 ﾁｬｯｸ 開
      ANI     Y10CB  ; SV39 芯金 後退
      ANI     Y10C5  ; SV12 ｻｲﾄﾞﾌﾞｰｽﾀ- 後退
      ANI     Y10C9  ; SV20 ﾊﾟｲﾌﾟ受け 下降
      INV
      ORB
      ANI     M7780  ; 強制出力中
      OR      B1D0  ; SV1油圧ﾎﾟﾝﾌﾟｵﾝﾛｰﾄﾞ
      ANB
      ANI     Y95  ; SV2 油圧ﾎﾟﾝﾌﾟｳｫｰﾐﾝｸﾞｱｯﾌﾟ
      OUT     Y94  ; SV1 油圧ﾎﾟﾝﾌﾟｵﾝﾛｰﾄﾞ
; 
      P2902
54    LD      SM400  ; 常時 ON
      MPS
      LD      M206  ; ﾋﾈﾘ_正転要求
      AND     T26  ; 捻りﾌﾞﾚｰｷ解除確認時間
      LD      M234  ; ﾋﾈﾘ_寸動用ﾌﾞﾚｰｷ開
      AND     Y13C4  ; SV29 ﾋﾈﾘ 減速正転
      ANI     M7012  ; D70=120ﾌﾗﾝｼﾞ穴検出手動
      ANI     M7016  ; D70=160再ﾌﾗﾝｼﾞ穴検出手動
      ORB
      AND     M200  ; ﾋﾈﾘ_正転IL
      ANI     M1  ; 一時停止中
      OR      B1AB  ; SV29ﾊﾟｲﾌﾟ捻り減速正転
      ANB
      ANI     Y13C5  ; SV30 ﾋﾈﾘ 減速逆転
      OUT     Y13C4  ; SV29 ﾋﾈﾘ 減速正転
      MPP
      LD      M206  ; ﾋﾈﾘ_正転要求
      AND     T26  ; 捻りﾌﾞﾚｰｷ解除確認時間
      ANI     M1927  ; ﾌﾗﾝｼﾞ穴検出D86=017_捻り正転
      ANI     M1722  ; 捻り原点復帰原点復帰減速正転
      LDI     M209  ; ﾋﾈﾘ_正転減速位置
      LDI     M7012  ; D70=120ﾌﾗﾝｼﾞ穴検出手動
      LDI     L101  ; 寸動選択_TB
      ANI     X1020  ; [ﾍﾟﾝﾀﾞﾝﾄ] 4PB1 ﾋﾈﾘ 正転
      ANI     X1007  ; 2PBL8 ﾋﾈﾘ 正転
      ORB
      ANB
      LD      L116  ; 手動選択_ﾗﾝﾌﾟ
      LD      X1020  ; [ﾍﾟﾝﾀﾞﾝﾄ] 4PB1 ﾋﾈﾘ 正転
      OR      X1007  ; 2PBL8 ﾋﾈﾘ 正転
      ANB
      ORB
      ANB
      AND     M200  ; ﾋﾈﾘ_正転IL
      ANI     M1  ; 一時停止中
      OR      B1A9  ; SV27ﾊﾟｲﾌﾟ捻り正転
      ANB
      ANI     Y13C3  ; SV28 ﾋﾈﾘ 逆転
      OUT     Y13C2  ; SV27 ﾋﾈﾘ 正転
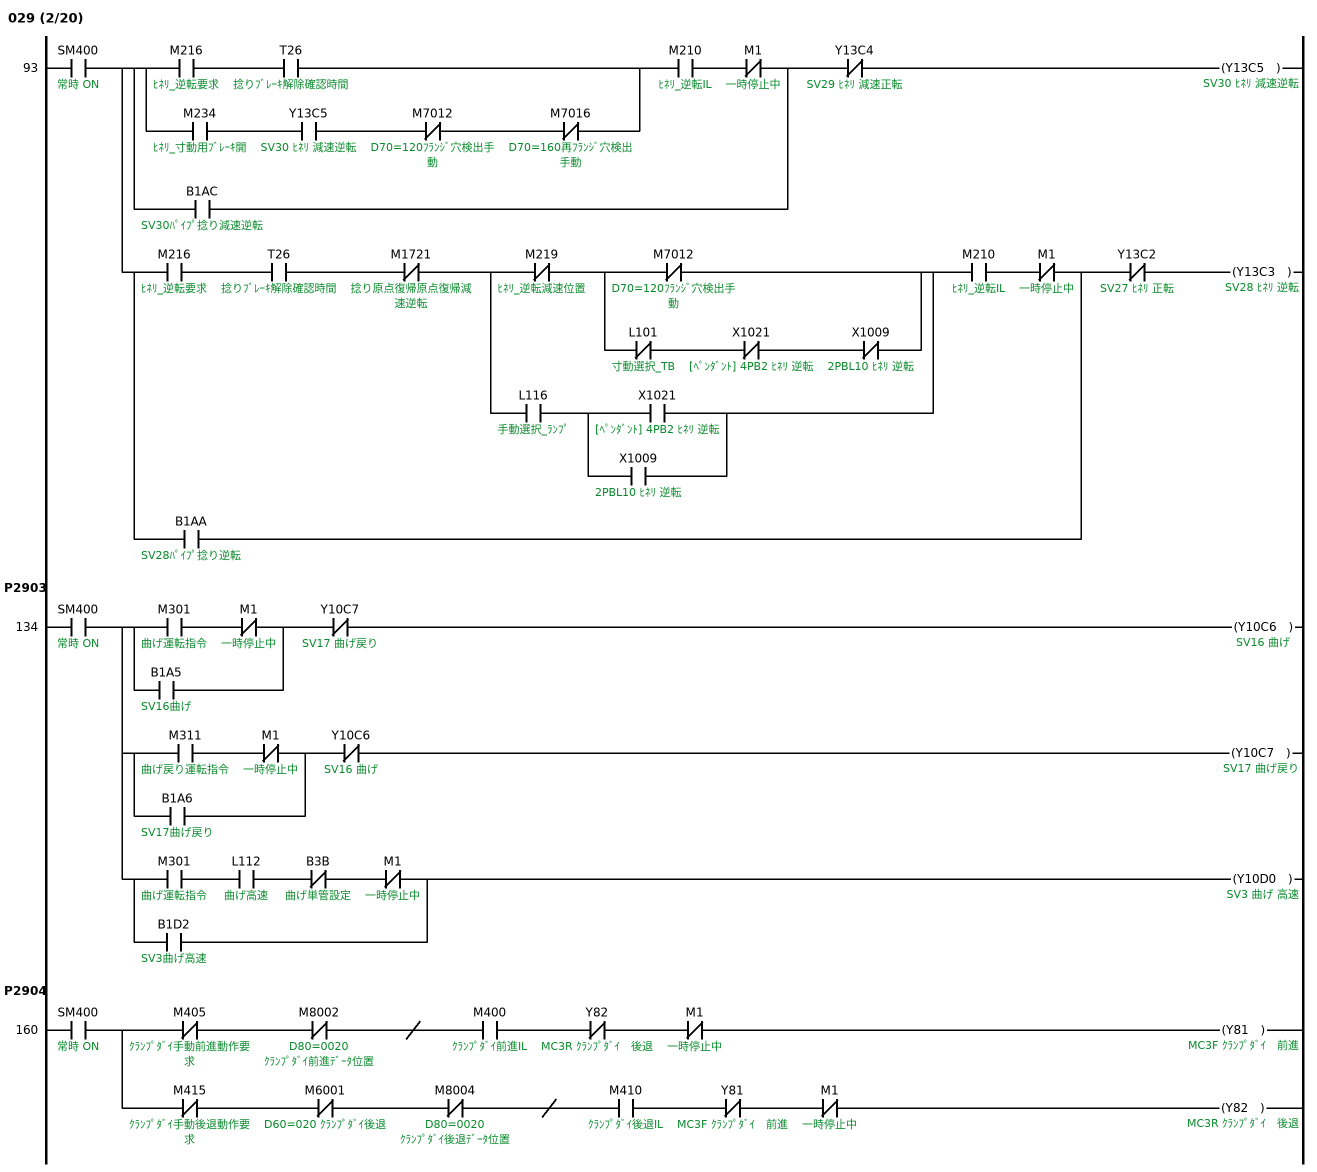
93    LD      SM400  ; 常時 ON
      MPS
      LD      M216  ; ﾋﾈﾘ_逆転要求
      AND     T26  ; 捻りﾌﾞﾚｰｷ解除確認時間
      LD      M234  ; ﾋﾈﾘ_寸動用ﾌﾞﾚｰｷ開
      AND     Y13C5  ; SV30 ﾋﾈﾘ 減速逆転
      ANI     M7012  ; D70=120ﾌﾗﾝｼﾞ穴検出手動
      ANI     M7016  ; D70=160再ﾌﾗﾝｼﾞ穴検出手動
      ORB
      AND     M210  ; ﾋﾈﾘ_逆転IL
      ANI     M1  ; 一時停止中
      OR      B1AC  ; SV30ﾊﾟｲﾌﾟ捻り減速逆転
      ANB
      ANI     Y13C4  ; SV29 ﾋﾈﾘ 減速正転
      OUT     Y13C5  ; SV30 ﾋﾈﾘ 減速逆転
      MPP
      LD      M216  ; ﾋﾈﾘ_逆転要求
      AND     T26  ; 捻りﾌﾞﾚｰｷ解除確認時間
      ANI     M1721  ; 捻り原点復帰原点復帰減速逆転
      LDI     M219  ; ﾋﾈﾘ_逆転減速位置
      LDI     M7012  ; D70=120ﾌﾗﾝｼﾞ穴検出手動
      LDI     L101  ; 寸動選択_TB
      ANI     X1021  ; [ﾍﾟﾝﾀﾞﾝﾄ] 4PB2 ﾋﾈﾘ 逆転
      ANI     X1009  ; 2PBL10 ﾋﾈﾘ 逆転
      ORB
      ANB
      LD      L116  ; 手動選択_ﾗﾝﾌﾟ
      LD      X1021  ; [ﾍﾟﾝﾀﾞﾝﾄ] 4PB2 ﾋﾈﾘ 逆転
      OR      X1009  ; 2PBL10 ﾋﾈﾘ 逆転
      ANB
      ORB
      ANB
      AND     M210  ; ﾋﾈﾘ_逆転IL
      ANI     M1  ; 一時停止中
      OR      B1AA  ; SV28ﾊﾟｲﾌﾟ捻り逆転
      ANB
      ANI     Y13C2  ; SV27 ﾋﾈﾘ 正転
      OUT     Y13C3  ; SV28 ﾋﾈﾘ 逆転
; 
      P2903
134   LD      SM400  ; 常時 ON
      MPS
      LD      M301  ; 曲げ運転指令
      ANI     M1  ; 一時停止中
      OR      B1A5  ; SV16曲げ
      ANB
      ANI     Y10C7  ; SV17 曲げ戻り
      OUT     Y10C6  ; SV16 曲げ
      MRD
      LD      M311  ; 曲げ戻り運転指令
      ANI     M1  ; 一時停止中
      OR      B1A6  ; SV17曲げ戻り
      ANB
      ANI     Y10C6  ; SV16 曲げ
      OUT     Y10C7  ; SV17 曲げ戻り
      MPP
      LD      M301  ; 曲げ運転指令
      AND     L112  ; 曲げ高速
      ANI     B3B  ; 曲げ単管設定
      ANI     M1  ; 一時停止中
      OR      B1D2  ; SV3曲げ高速
      ANB
      OUT     Y10D0  ; SV3 曲げ 高速
; 
      P2904
160   LD      SM400  ; 常時 ON
      MPS
      ANI     M405  ; ｸﾗﾝﾌﾟﾀﾞｲ手動前進動作要求
      ANI     M8002  ; D80=0020 ｸﾗﾝﾌﾟﾀﾞｲ前進ﾃﾞｰﾀ位置
      INV
      AND     M400  ; ｸﾗﾝﾌﾟﾀﾞｲ前進IL
      ANI     Y82  ; MC3R ｸﾗﾝﾌﾟﾀﾞｲ　後退
      ANI     M1  ; 一時停止中
      OUT     Y81  ; MC3F ｸﾗﾝﾌﾟﾀﾞｲ　前進
      MPP
      ANI     M415  ; ｸﾗﾝﾌﾟﾀﾞｲ手動後退動作要求
      ANI     M6001  ; D60=020 ｸﾗﾝﾌﾟﾀﾞｲ後退
      ANI     M8004  ; D80=0020 ｸﾗﾝﾌﾟﾀﾞｲ後退ﾃﾞｰﾀ位置
      INV
      AND     M410  ; ｸﾗﾝﾌﾟﾀﾞｲ後退IL
      ANI     Y81  ; MC3F ｸﾗﾝﾌﾟﾀﾞｲ　前進
      ANI     M1  ; 一時停止中
      OUT     Y82  ; MC3R ｸﾗﾝﾌﾟﾀﾞｲ　後退
; 
      P2905
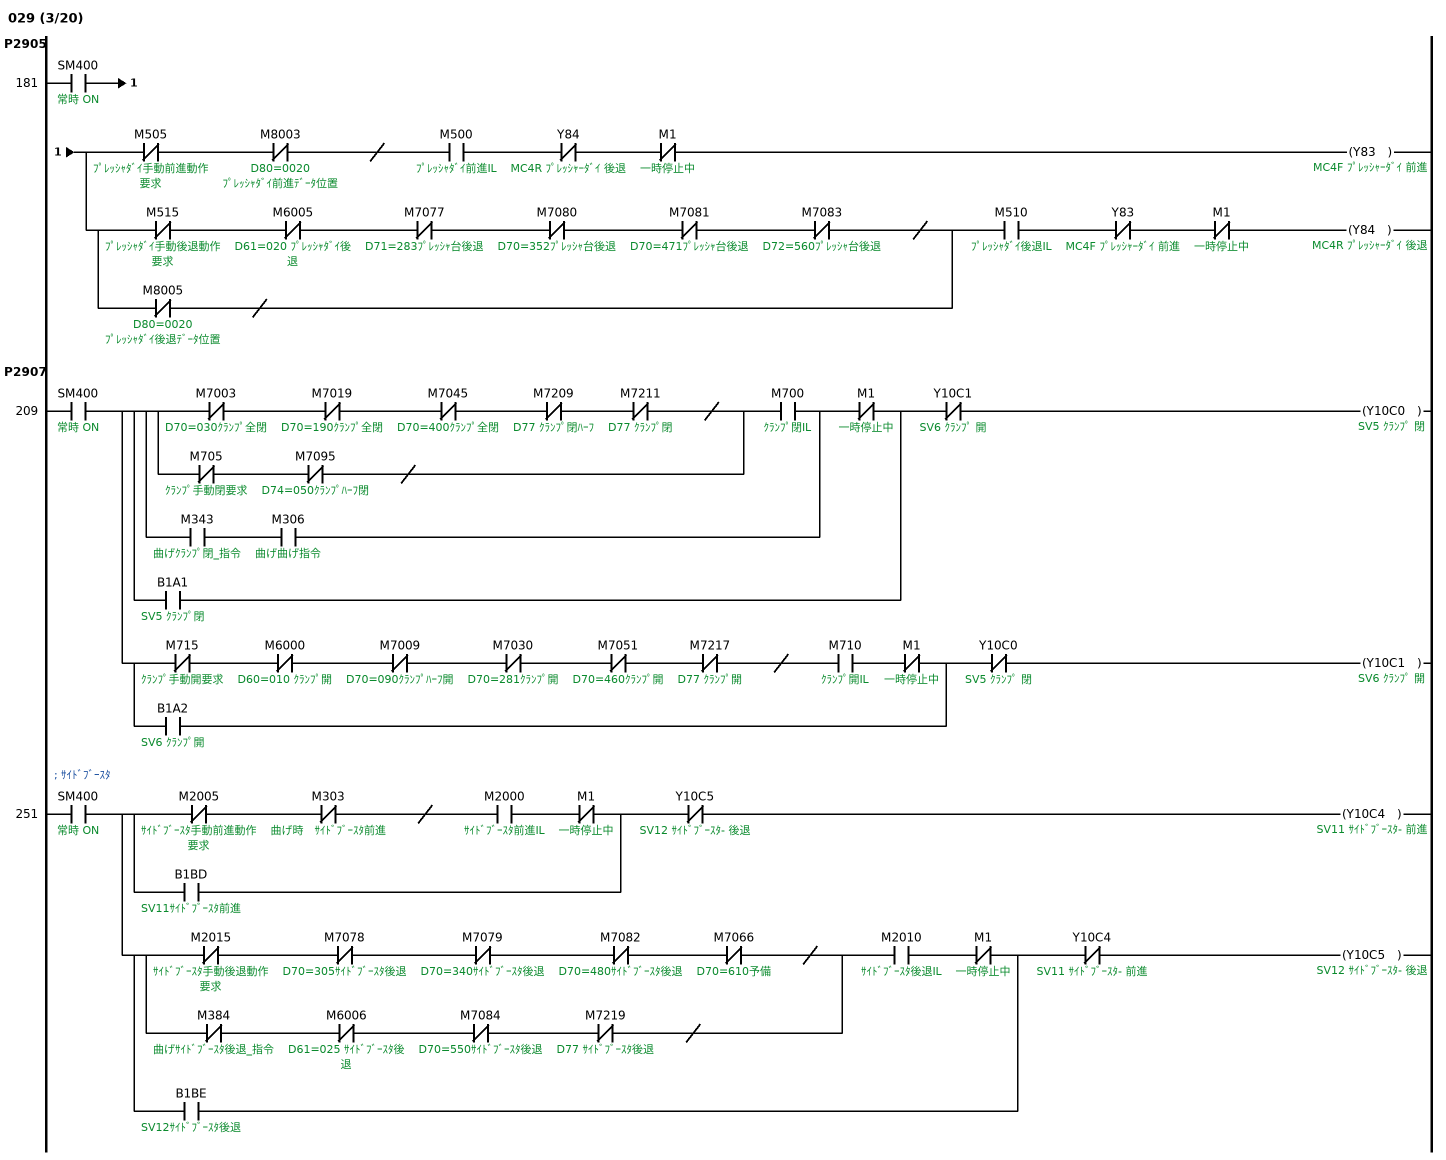
181   LD      SM400  ; 常時 ON
      MPS
      ANI     M505  ; ﾌﾟﾚｯｼｬﾀﾞｲ手動前進動作要求
      ANI     M8003  ; D80=0020 ﾌﾟﾚｯｼｬﾀﾞｲ前進ﾃﾞｰﾀ位置
      INV
      AND     M500  ; ﾌﾟﾚｯｼｬﾀﾞｲ前進IL
      ANI     Y84  ; MC4R ﾌﾟﾚｯｼｬｰﾀﾞｲ 後退
      ANI     M1  ; 一時停止中
      OUT     Y83  ; MC4F ﾌﾟﾚｯｼｬｰﾀﾞｲ 前進
      MPP
      LDI     M515  ; ﾌﾟﾚｯｼｬﾀﾞｲ手動後退動作要求
      ANI     M6005  ; D61=020 ﾌﾟﾚｯｼｬﾀﾞｲ後退
      ANI     M7077  ; D71=283ﾌﾟﾚｯｼｬ台後退
      ANI     M7080  ; D70=352ﾌﾟﾚｯｼｬ台後退
      ANI     M7081  ; D70=471ﾌﾟﾚｯｼｬ台後退
      ANI     M7083  ; D72=560ﾌﾟﾚｯｼｬ台後退
      INV
      LDI     M8005  ; D80=0020 ﾌﾟﾚｯｼｬﾀﾞｲ後退ﾃﾞｰﾀ位置
      INV
      ORB
      ANB
      AND     M510  ; ﾌﾟﾚｯｼｬﾀﾞｲ後退IL
      ANI     Y83  ; MC4F ﾌﾟﾚｯｼｬｰﾀﾞｲ 前進
      ANI     M1  ; 一時停止中
      OUT     Y84  ; MC4R ﾌﾟﾚｯｼｬｰﾀﾞｲ 後退
; 
      P2907
209   LD      SM400  ; 常時 ON
      MPS
      LDI     M7003  ; D70=030ｸﾗﾝﾌﾟ全閉
      ANI     M7019  ; D70=190ｸﾗﾝﾌﾟ全閉
      ANI     M7045  ; D70=400ｸﾗﾝﾌﾟ全閉
      ANI     M7209  ; D77 ｸﾗﾝﾌﾟ閉ﾊｰﾌ
      ANI     M7211  ; D77 ｸﾗﾝﾌﾟ閉
      INV
      LDI     M705  ; ｸﾗﾝﾌﾟ手動閉要求
      ANI     M7095  ; D74=050ｸﾗﾝﾌﾟﾊｰﾌ閉
      INV
      ORB
      AND     M700  ; ｸﾗﾝﾌﾟ閉IL
      LD      M343  ; 曲げｸﾗﾝﾌﾟ閉_指令
      AND     M306  ; 曲げ曲げ指令
      ORB
      ANI     M1  ; 一時停止中
      OR      B1A1  ; SV5 ｸﾗﾝﾌﾟ閉
      ANB
      ANI     Y10C1  ; SV6 ｸﾗﾝﾌﾟ 開
      OUT     Y10C0  ; SV5 ｸﾗﾝﾌﾟ 閉
      MPP
      LDI     M715  ; ｸﾗﾝﾌﾟ手動開要求
      ANI     M6000  ; D60=010 ｸﾗﾝﾌﾟ開
      ANI     M7009  ; D70=090ｸﾗﾝﾌﾟﾊｰﾌ開
      ANI     M7030  ; D70=281ｸﾗﾝﾌﾟ開
      ANI     M7051  ; D70=460ｸﾗﾝﾌﾟ開
      ANI     M7217  ; D77 ｸﾗﾝﾌﾟ開
      INV
      AND     M710  ; ｸﾗﾝﾌﾟ開IL
      ANI     M1  ; 一時停止中
      OR      B1A2  ; SV6 ｸﾗﾝﾌﾟ開
      ANB
      ANI     Y10C0  ; SV5 ｸﾗﾝﾌﾟ 閉
      OUT     Y10C1  ; SV6 ｸﾗﾝﾌﾟ 開
; ｻｲﾄﾞﾌﾞｰｽﾀ
251   LD      SM400  ; 常時 ON
      MPS
      LDI     M2005  ; ｻｲﾄﾞﾌﾞｰｽﾀ手動前進動作要求
      ANI     M303  ; 曲げ時　ｻｲﾄﾞﾌﾞｰｽﾀ前進
      INV
      AND     M2000  ; ｻｲﾄﾞﾌﾞｰｽﾀ前進IL
      ANI     M1  ; 一時停止中
      OR      B1BD  ; SV11ｻｲﾄﾞﾌﾞｰｽﾀ前進
      ANB
      ANI     Y10C5  ; SV12 ｻｲﾄﾞﾌﾞｰｽﾀ- 後退
      OUT     Y10C4  ; SV11 ｻｲﾄﾞﾌﾞｰｽﾀ- 前進
      MPP
      LDI     M2015  ; ｻｲﾄﾞﾌﾞｰｽﾀ手動後退動作要求
      ANI     M7078  ; D70=305ｻｲﾄﾞﾌﾞｰｽﾀ後退
      ANI     M7079  ; D70=340ｻｲﾄﾞﾌﾞｰｽﾀ後退
      ANI     M7082  ; D70=480ｻｲﾄﾞﾌﾞｰｽﾀ後退
      ANI     M7066  ; D70=610予備
      INV
      LDI     M384  ; 曲げｻｲﾄﾞﾌﾞｰｽﾀ後退_指令
      ANI     M6006  ; D61=025 ｻｲﾄﾞﾌﾞｰｽﾀ後退
      ANI     M7084  ; D70=550ｻｲﾄﾞﾌﾞｰｽﾀ後退
      ANI     M7219  ; D77 ｻｲﾄﾞﾌﾞｰｽﾀ後退
      INV
      ORB
      AND     M2010  ; ｻｲﾄﾞﾌﾞｰｽﾀ後退IL
      ANI     M1  ; 一時停止中
      OR      B1BE  ; SV12ｻｲﾄﾞﾌﾞｰｽﾀ後退
      ANB
      ANI     Y10C4  ; SV11 ｻｲﾄﾞﾌﾞｰｽﾀ- 前進
      OUT     Y10C5  ; SV12 ｻｲﾄﾞﾌﾞｰｽﾀ- 後退
; 
      P2908
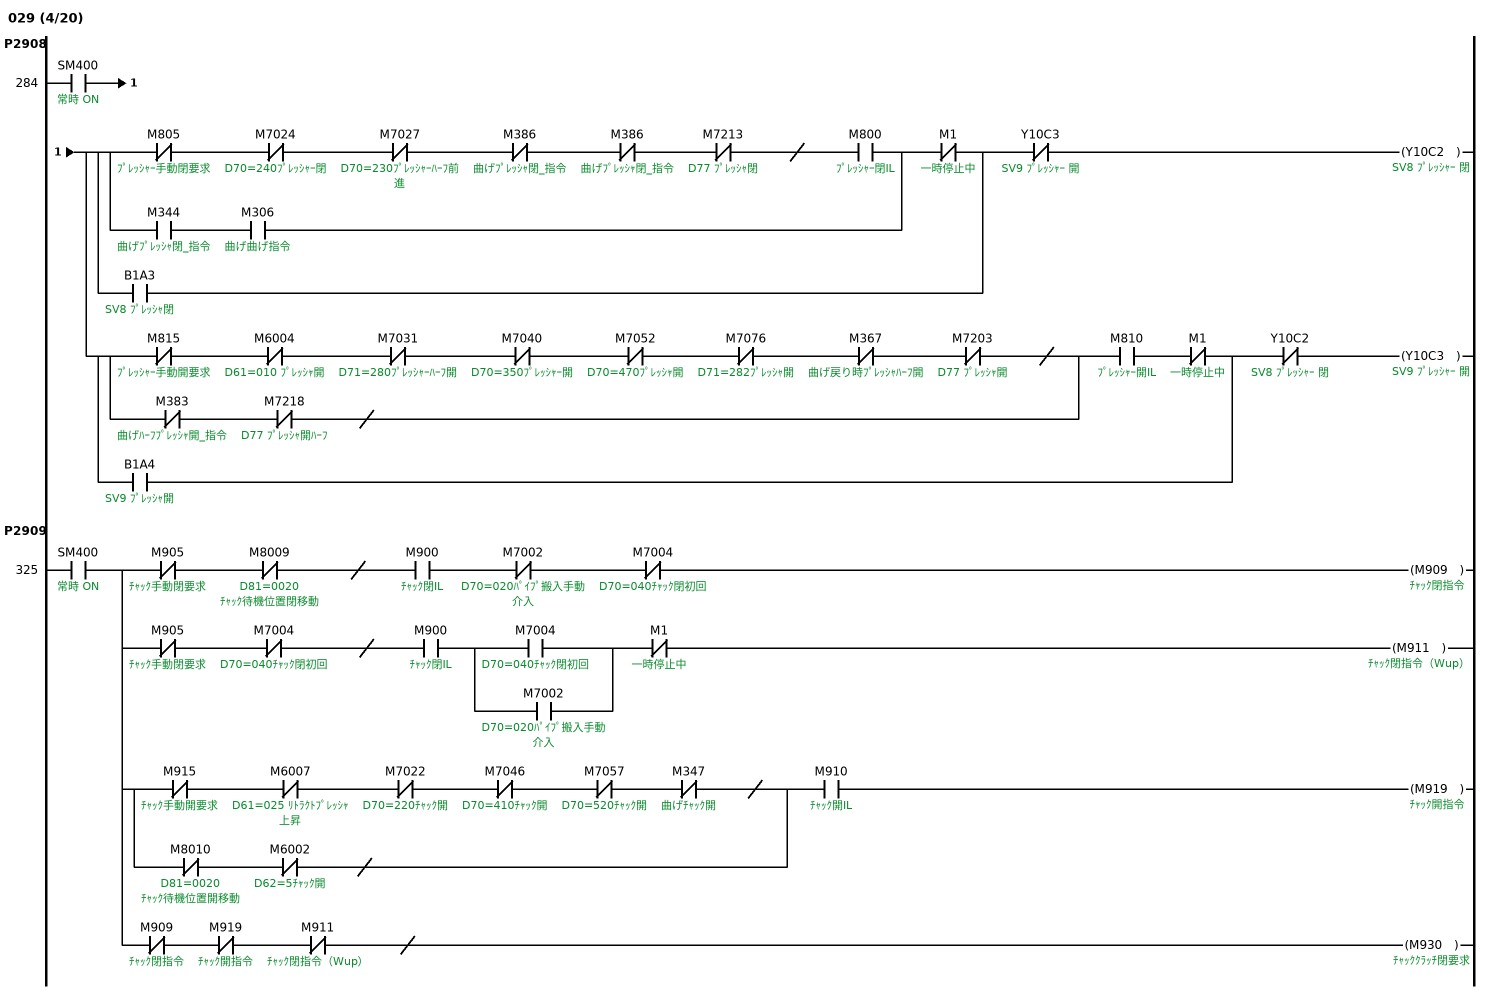
284   LD      SM400  ; 常時 ON
      MPS
      LDI     M805  ; ﾌﾟﾚｯｼｬｰ手動閉要求
      ANI     M7024  ; D70=240ﾌﾟﾚｯｼｬｰ閉
      ANI     M7027  ; D70=230ﾌﾟﾚｯｼｬｰﾊｰﾌ前進
      ANI     M386  ; 曲げﾌﾟﾚｯｼｬ閉_指令
      ANI     M386  ; 曲げﾌﾟﾚｯｼｬ閉_指令
      ANI     M7213  ; D77 ﾌﾟﾚｯｼｬ閉
      INV
      AND     M800  ; ﾌﾟﾚｯｼｬｰ閉IL
      LD      M344  ; 曲げﾌﾟﾚｯｼｬ閉_指令
      AND     M306  ; 曲げ曲げ指令
      ORB
      ANI     M1  ; 一時停止中
      OR      B1A3  ; SV8 ﾌﾟﾚｯｼｬ閉
      ANB
      ANI     Y10C3  ; SV9 ﾌﾟﾚｯｼｬｰ 開
      OUT     Y10C2  ; SV8 ﾌﾟﾚｯｼｬｰ 閉
      MPP
      LDI     M815  ; ﾌﾟﾚｯｼｬｰ手動開要求
      ANI     M6004  ; D61=010 ﾌﾟﾚｯｼｬ開
      ANI     M7031  ; D71=280ﾌﾟﾚｯｼｬｰﾊｰﾌ開
      ANI     M7040  ; D70=350ﾌﾟﾚｯｼｬｰ開
      ANI     M7052  ; D70=470ﾌﾟﾚｯｼｬ開
      ANI     M7076  ; D71=282ﾌﾟﾚｯｼｬ開
      ANI     M367  ; 曲げ戻り時ﾌﾟﾚｯｼｬﾊｰﾌ開
      ANI     M7203  ; D77 ﾌﾟﾚｯｼｬ開
      INV
      LDI     M383  ; 曲げﾊｰﾌﾌﾟﾚｯｼｬ開_指令
      ANI     M7218  ; D77 ﾌﾟﾚｯｼｬ開ﾊｰﾌ
      INV
      ORB
      AND     M810  ; ﾌﾟﾚｯｼｬｰ開IL
      ANI     M1  ; 一時停止中
      OR      B1A4  ; SV9 ﾌﾟﾚｯｼｬ開
      ANB
      ANI     Y10C2  ; SV8 ﾌﾟﾚｯｼｬｰ 閉
      OUT     Y10C3  ; SV9 ﾌﾟﾚｯｼｬｰ 開
; 
      P2909
325   LD      SM400  ; 常時 ON
      MPS
      ANI     M905  ; ﾁｬｯｸ手動閉要求
      ANI     M8009  ; D81=0020 ﾁｬｯｸ待機位置閉移動
      INV
      AND     M900  ; ﾁｬｯｸ閉IL
      ANI     M7002  ; D70=020ﾊﾟｲﾌﾟ搬入手動介入
      ANI     M7004  ; D70=040ﾁｬｯｸ閉初回
      OUT     M909  ; ﾁｬｯｸ閉指令
      MRD
      ANI     M905  ; ﾁｬｯｸ手動閉要求
      ANI     M7004  ; D70=040ﾁｬｯｸ閉初回
      INV
      AND     M900  ; ﾁｬｯｸ閉IL
      LD      M7004  ; D70=040ﾁｬｯｸ閉初回
      OR      M7002  ; D70=020ﾊﾟｲﾌﾟ搬入手動介入
      ANB
      ANI     M1  ; 一時停止中
      OUT     M911  ; ﾁｬｯｸ閉指令（Wup）
      MRD
      LDI     M915  ; ﾁｬｯｸ手動開要求
      ANI     M6007  ; D61=025 ﾘﾄﾗｸﾄﾌﾟﾚｯｼｬ上昇
      ANI     M7022  ; D70=220ﾁｬｯｸ開
      ANI     M7046  ; D70=410ﾁｬｯｸ開
      ANI     M7057  ; D70=520ﾁｬｯｸ開
      ANI     M347  ; 曲げﾁｬｯｸ開
      INV
      LDI     M8010  ; D81=0020 ﾁｬｯｸ待機位置開移動
      ANI     M6002  ; D62=5ﾁｬｯｸ開
      INV
      ORB
      ANB
      AND     M910  ; ﾁｬｯｸ開IL
      OUT     M919  ; ﾁｬｯｸ開指令
      MPP
      ANI     M909  ; ﾁｬｯｸ閉指令
      ANI     M919  ; ﾁｬｯｸ開指令
      ANI     M911  ; ﾁｬｯｸ閉指令（Wup）
      INV
      OUT     M930  ; ﾁｬｯｸｸﾗｯﾁ閉要求
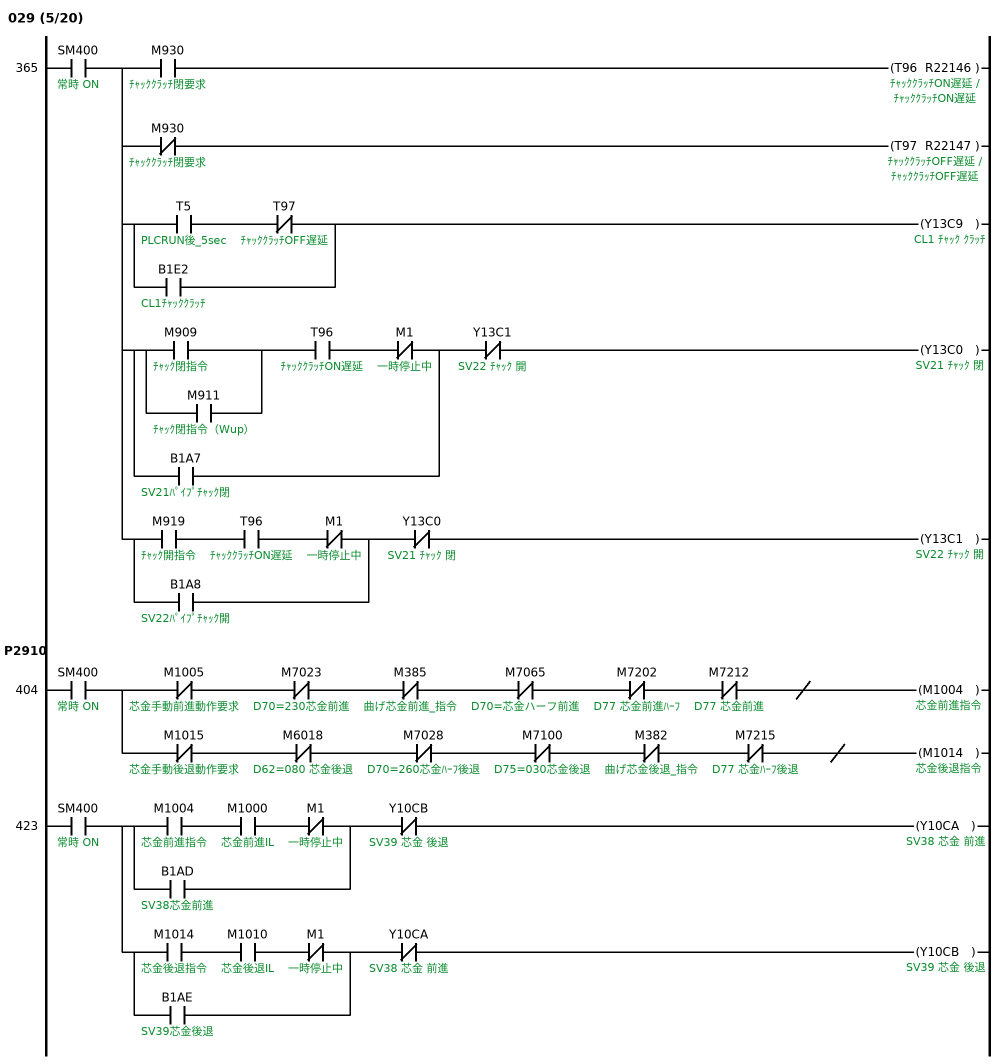
365   LD      SM400  ; 常時 ON
      MPS
      AND     M930  ; ﾁｬｯｸｸﾗｯﾁ閉要求
      OUT     T96 R22146  ; ﾁｬｯｸｸﾗｯﾁON遅延 / ﾁｬｯｸｸﾗｯﾁON遅延
      MRD
      ANI     M930  ; ﾁｬｯｸｸﾗｯﾁ閉要求
      OUT     T97 R22147  ; ﾁｬｯｸｸﾗｯﾁOFF遅延 / ﾁｬｯｸｸﾗｯﾁOFF遅延
      MRD
      LD      T5  ; PLCRUN後_5sec
      ANI     T97  ; ﾁｬｯｸｸﾗｯﾁOFF遅延
      OR      B1E2  ; CL1ﾁｬｯｸｸﾗｯﾁ
      ANB
      OUT     Y13C9  ; CL1 ﾁｬｯｸ ｸﾗｯﾁ
      MRD
      LD      M909  ; ﾁｬｯｸ閉指令
      OR      M911  ; ﾁｬｯｸ閉指令（Wup）
      AND     T96  ; ﾁｬｯｸｸﾗｯﾁON遅延
      ANI     M1  ; 一時停止中
      OR      B1A7  ; SV21ﾊﾟｲﾌﾟﾁｬｯｸ閉
      ANB
      ANI     Y13C1  ; SV22 ﾁｬｯｸ 開
      OUT     Y13C0  ; SV21 ﾁｬｯｸ 閉
      MPP
      LD      M919  ; ﾁｬｯｸ開指令
      AND     T96  ; ﾁｬｯｸｸﾗｯﾁON遅延
      ANI     M1  ; 一時停止中
      OR      B1A8  ; SV22ﾊﾟｲﾌﾟﾁｬｯｸ開
      ANB
      ANI     Y13C0  ; SV21 ﾁｬｯｸ 閉
      OUT     Y13C1  ; SV22 ﾁｬｯｸ 開
; 
      P2910
404   LD      SM400  ; 常時 ON
      MPS
      ANI     M1005  ; 芯金手動前進動作要求
      ANI     M7023  ; D70=230芯金前進
      ANI     M385  ; 曲げ芯金前進_指令
      ANI     M7065  ; D70=芯金ハーフ前進
      ANI     M7202  ; D77 芯金前進ﾊｰﾌ
      ANI     M7212  ; D77 芯金前進
      INV
      OUT     M1004  ; 芯金前進指令
      MPP
      ANI     M1015  ; 芯金手動後退動作要求
      ANI     M6018  ; D62=080 芯金後退
      ANI     M7028  ; D70=260芯金ﾊｰﾌ後退
      ANI     M7100  ; D75=030芯金後退
      ANI     M382  ; 曲げ芯金後退_指令
      ANI     M7215  ; D77 芯金ﾊｰﾌ後退
      INV
      OUT     M1014  ; 芯金後退指令
423   LD      SM400  ; 常時 ON
      MPS
      LD      M1004  ; 芯金前進指令
      AND     M1000  ; 芯金前進IL
      ANI     M1  ; 一時停止中
      OR      B1AD  ; SV38芯金前進
      ANB
      ANI     Y10CB  ; SV39 芯金 後退
      OUT     Y10CA  ; SV38 芯金 前進
      MPP
      LD      M1014  ; 芯金後退指令
      AND     M1010  ; 芯金後退IL
      ANI     M1  ; 一時停止中
      OR      B1AE  ; SV39芯金後退
      ANB
      ANI     Y10CA  ; SV38 芯金 前進
      OUT     Y10CB  ; SV39 芯金 後退
; 
      P2913
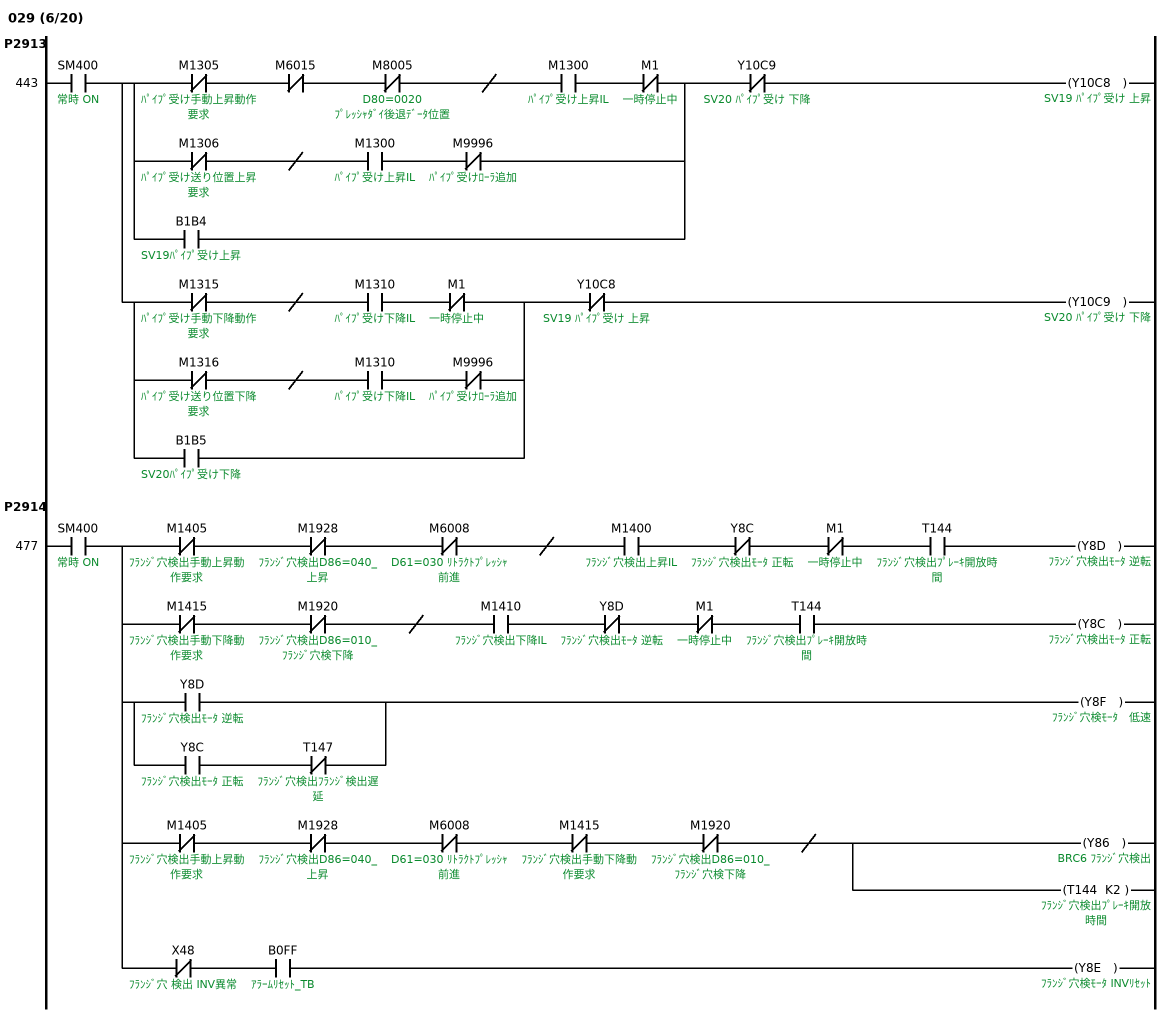
443   LD      SM400  ; 常時 ON
      MPS
      LDI     M1305  ; ﾊﾟｲﾌﾟ受け手動上昇動作要求
      ANI     M6015
      ANI     M8005  ; D80=0020 ﾌﾟﾚｯｼｬﾀﾞｲ後退ﾃﾞｰﾀ位置
      INV
      AND     M1300  ; ﾊﾟｲﾌﾟ受け上昇IL
      ANI     M1  ; 一時停止中
      LDI     M1306  ; ﾊﾟｲﾌﾟ受け送り位置上昇要求
      INV
      AND     M1300  ; ﾊﾟｲﾌﾟ受け上昇IL
      ANI     M9996  ; ﾊﾟｲﾌﾟ受けﾛｰﾗ追加
      ORB
      OR      B1B4  ; SV19ﾊﾟｲﾌﾟ受け上昇
      ANB
      ANI     Y10C9  ; SV20 ﾊﾟｲﾌﾟ受け 下降
      OUT     Y10C8  ; SV19 ﾊﾟｲﾌﾟ受け 上昇
      MPP
      LDI     M1315  ; ﾊﾟｲﾌﾟ受け手動下降動作要求
      INV
      AND     M1310  ; ﾊﾟｲﾌﾟ受け下降IL
      ANI     M1  ; 一時停止中
      LDI     M1316  ; ﾊﾟｲﾌﾟ受け送り位置下降要求
      INV
      AND     M1310  ; ﾊﾟｲﾌﾟ受け下降IL
      ANI     M9996  ; ﾊﾟｲﾌﾟ受けﾛｰﾗ追加
      ORB
      OR      B1B5  ; SV20ﾊﾟｲﾌﾟ受け下降
      ANB
      ANI     Y10C8  ; SV19 ﾊﾟｲﾌﾟ受け 上昇
      OUT     Y10C9  ; SV20 ﾊﾟｲﾌﾟ受け 下降
; 
      P2914
477   LD      SM400  ; 常時 ON
      MPS
      ANI     M1405  ; ﾌﾗﾝｼﾞ穴検出手動上昇動作要求
      ANI     M1928  ; ﾌﾗﾝｼﾞ穴検出D86=040_上昇
      ANI     M6008  ; D61=030 ﾘﾄﾗｸﾄﾌﾟﾚｯｼｬ前進
      INV
      AND     M1400  ; ﾌﾗﾝｼﾞ穴検出上昇IL
      ANI     Y8C  ; ﾌﾗﾝｼﾞ穴検出ﾓｰﾀ 正転
      ANI     M1  ; 一時停止中
      AND     T144  ; ﾌﾗﾝｼﾞ穴検出ﾌﾟﾚｰｷ開放時間
      OUT     Y8D  ; ﾌﾗﾝｼﾞ穴検出ﾓｰﾀ 逆転
      MRD
      ANI     M1415  ; ﾌﾗﾝｼﾞ穴検出手動下降動作要求
      ANI     M1920  ; ﾌﾗﾝｼﾞ穴検出D86=010_ﾌﾗﾝｼﾞ穴検下降
      INV
      AND     M1410  ; ﾌﾗﾝｼﾞ穴検出下降IL
      ANI     Y8D  ; ﾌﾗﾝｼﾞ穴検出ﾓｰﾀ 逆転
      ANI     M1  ; 一時停止中
      AND     T144  ; ﾌﾗﾝｼﾞ穴検出ﾌﾟﾚｰｷ開放時間
      OUT     Y8C  ; ﾌﾗﾝｼﾞ穴検出ﾓｰﾀ 正転
      MRD
      LD      Y8D  ; ﾌﾗﾝｼﾞ穴検出ﾓｰﾀ 逆転
      LD      Y8C  ; ﾌﾗﾝｼﾞ穴検出ﾓｰﾀ 正転
      ANI     T147  ; ﾌﾗﾝｼﾞ穴検出ﾌﾗﾝｼﾞ検出遅延
      ORB
      ANB
      OUT     Y8F  ; ﾌﾗﾝｼﾞ穴検ﾓｰﾀ　低速
      MRD
      ANI     M1405  ; ﾌﾗﾝｼﾞ穴検出手動上昇動作要求
      ANI     M1928  ; ﾌﾗﾝｼﾞ穴検出D86=040_上昇
      ANI     M6008  ; D61=030 ﾘﾄﾗｸﾄﾌﾟﾚｯｼｬ前進
      ANI     M1415  ; ﾌﾗﾝｼﾞ穴検出手動下降動作要求
      ANI     M1920  ; ﾌﾗﾝｼﾞ穴検出D86=010_ﾌﾗﾝｼﾞ穴検下降
      INV
      OUT     Y86  ; BRC6 ﾌﾗﾝｼﾞ穴検出
      OUT     T144 K2  ; ﾌﾗﾝｼﾞ穴検出ﾌﾟﾚｰｷ開放時間
      MPP
      ANI     X48  ; ﾌﾗﾝｼﾞ穴 検出 INV異常
      AND     B0FF  ; ｱﾗｰﾑﾘｾｯﾄ_TB
      OUT     Y8E  ; ﾌﾗﾝｼﾞ穴検ﾓｰﾀ INVﾘｾｯﾄ
; 
      P2915
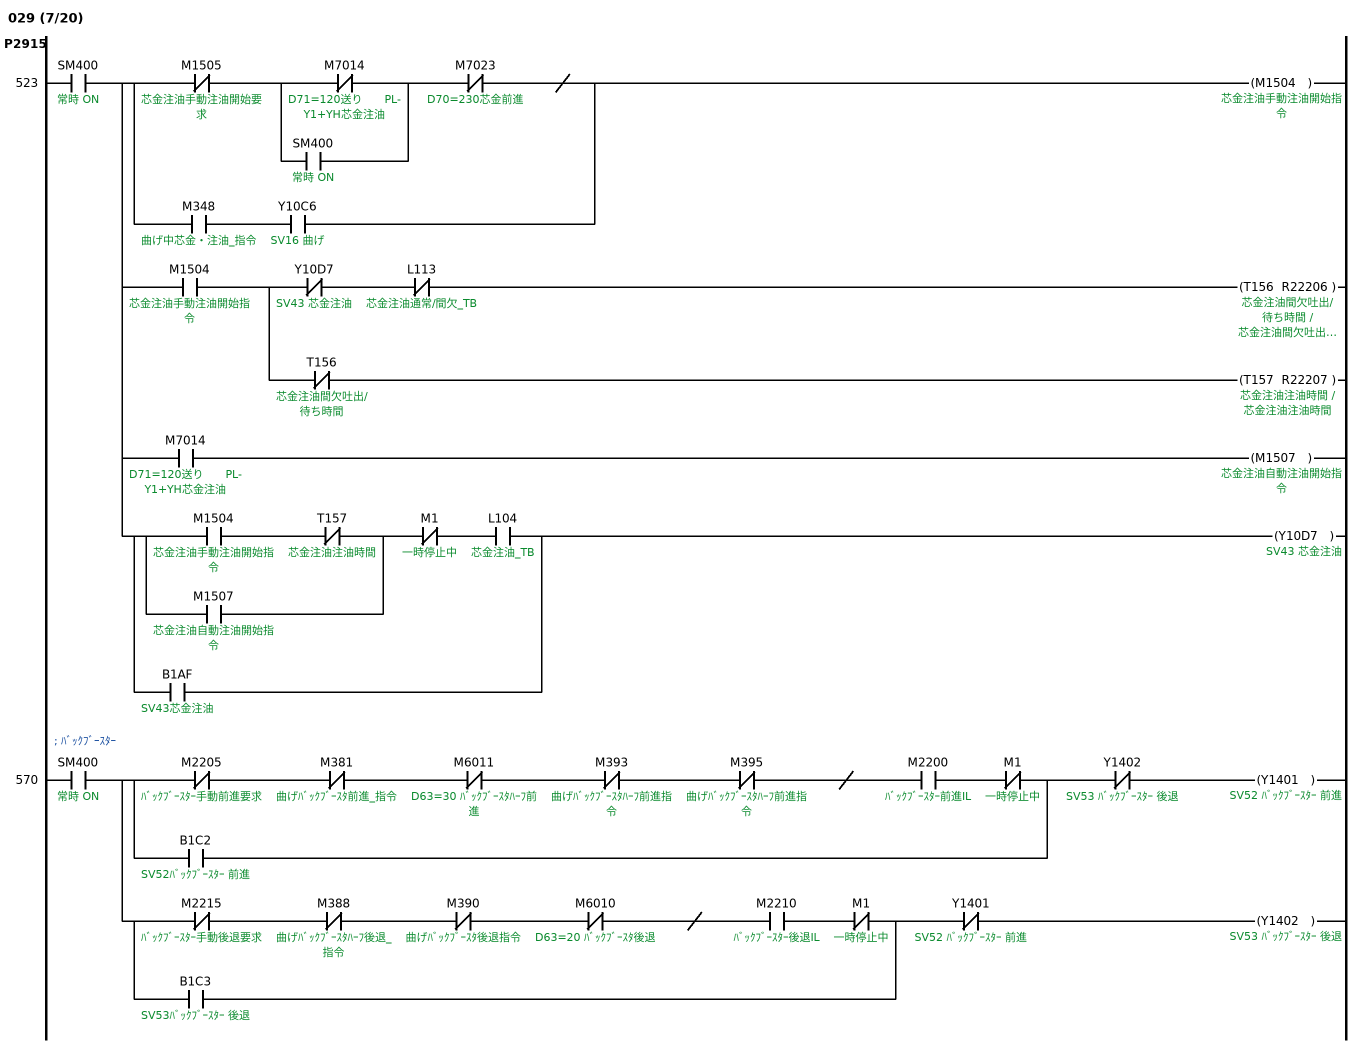
523   LD      SM400  ; 常時 ON
      MPS
      LDI     M1505  ; 芯金注油手動注油開始要求
      LDI     M7014  ; D71=120送り　　PL-Y1+YH芯金注油
      OR      SM400  ; 常時 ON
      ANB
      ANI     M7023  ; D70=230芯金前進
      INV
      LD      M348  ; 曲げ中芯金・注油_指令
      AND     Y10C6  ; SV16 曲げ
      ORB
      ANB
      OUT     M1504  ; 芯金注油手動注油開始指令
      MRD
      AND     M1504  ; 芯金注油手動注油開始指令
      MPS
      ANI     Y10D7  ; SV43 芯金注油
      ANI     L113  ; 芯金注油通常/間欠_TB
      OUT     T156 R22206  ; 芯金注油間欠吐出/待ち時間 / 芯金注油間欠吐出/待ち時間
      MPP
      ANI     T156  ; 芯金注油間欠吐出/待ち時間
      OUT     T157 R22207  ; 芯金注油注油時間 / 芯金注油注油時間
      MRD
      AND     M7014  ; D71=120送り　　PL-Y1+YH芯金注油
      OUT     M1507  ; 芯金注油自動注油開始指令
      MPP
      LD      M1504  ; 芯金注油手動注油開始指令
      ANI     T157  ; 芯金注油注油時間
      OR      M1507  ; 芯金注油自動注油開始指令
      ANI     M1  ; 一時停止中
      AND     L104  ; 芯金注油_TB
      OR      B1AF  ; SV43芯金注油
      ANB
      OUT     Y10D7  ; SV43 芯金注油
; ﾊﾞｯｸﾌﾞｰｽﾀｰ
570   LD      SM400  ; 常時 ON
      MPS
      LDI     M2205  ; ﾊﾞｯｸﾌﾞｰｽﾀｰ手動前進要求
      ANI     M381  ; 曲げﾊﾞｯｸﾌﾞｰｽﾀ前進_指令
      ANI     M6011  ; D63=30 ﾊﾞｯｸﾌﾞｰｽﾀﾊｰﾌ前進
      ANI     M393  ; 曲げﾊﾞｯｸﾌﾞｰｽﾀﾊｰﾌ前進指令
      ANI     M395  ; 曲げﾊﾞｯｸﾌﾞｰｽﾀﾊｰﾌ前進指令
      INV
      AND     M2200  ; ﾊﾞｯｸﾌﾞｰｽﾀｰ前進IL
      ANI     M1  ; 一時停止中
      OR      B1C2  ; SV52ﾊﾞｯｸﾌﾞｰｽﾀｰ 前進
      ANB
      ANI     Y1402  ; SV53 ﾊﾞｯｸﾌﾞｰｽﾀｰ 後退
      OUT     Y1401  ; SV52 ﾊﾞｯｸﾌﾞｰｽﾀｰ 前進
      MPP
      LDI     M2215  ; ﾊﾞｯｸﾌﾞｰｽﾀｰ手動後退要求
      ANI     M388  ; 曲げﾊﾞｯｸﾌﾞｰｽﾀﾊｰﾌ後退_指令
      ANI     M390  ; 曲げﾊﾞｯｸﾌﾞｰｽﾀ後退指令
      ANI     M6010  ; D63=20 ﾊﾞｯｸﾌﾞｰｽﾀ後退
      INV
      AND     M2210  ; ﾊﾞｯｸﾌﾞｰｽﾀｰ後退IL
      ANI     M1  ; 一時停止中
      OR      B1C3  ; SV53ﾊﾞｯｸﾌﾞｰｽﾀｰ 後退
      ANB
      ANI     Y1401  ; SV52 ﾊﾞｯｸﾌﾞｰｽﾀｰ 前進
      OUT     Y1402  ; SV53 ﾊﾞｯｸﾌﾞｰｽﾀｰ 後退
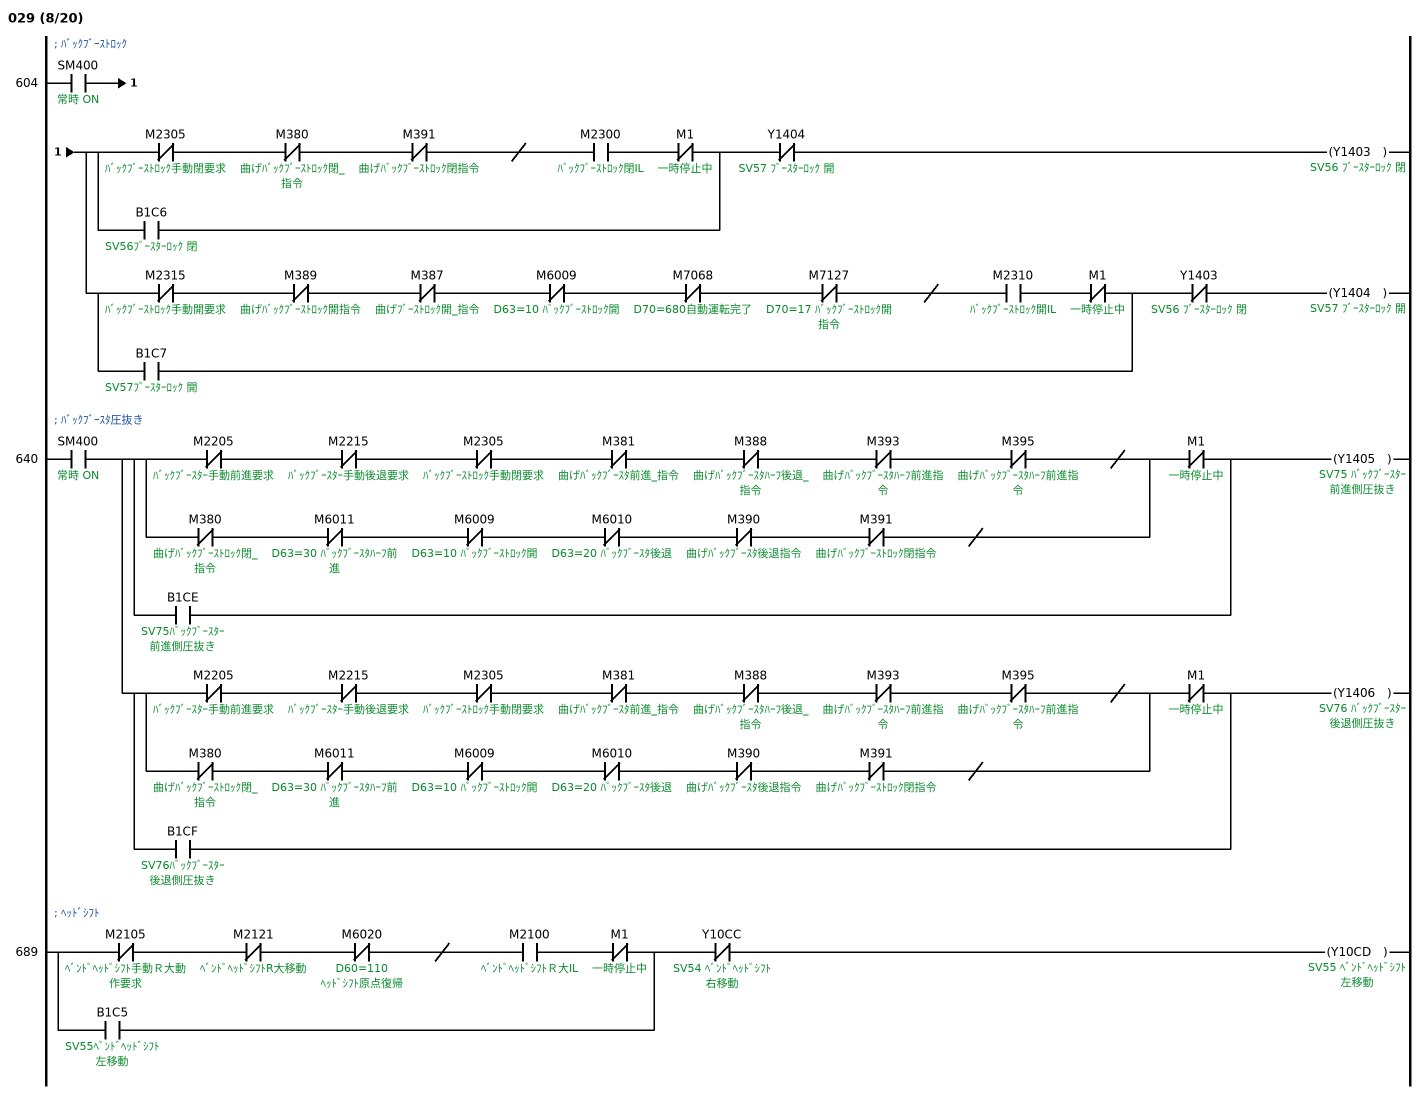
; ﾊﾞｯｸﾌﾞｰｽﾄﾛｯｸ
604   LD      SM400  ; 常時 ON
      MPS
      LDI     M2305  ; ﾊﾞｯｸﾌﾞｰｽﾄﾛｯｸ手動閉要求
      ANI     M380  ; 曲げﾊﾞｯｸﾌﾞｰｽﾄﾛｯｸ閉_指令
      ANI     M391  ; 曲げﾊﾞｯｸﾌﾞｰｽﾄﾛｯｸ閉指令
      INV
      AND     M2300  ; ﾊﾞｯｸﾌﾞｰｽﾄﾛｯｸ閉IL
      ANI     M1  ; 一時停止中
      OR      B1C6  ; SV56ﾌﾞｰｽﾀｰﾛｯｸ 閉
      ANB
      ANI     Y1404  ; SV57 ﾌﾞｰｽﾀｰﾛｯｸ 開
      OUT     Y1403  ; SV56 ﾌﾞｰｽﾀｰﾛｯｸ 閉
      MPP
      LDI     M2315  ; ﾊﾞｯｸﾌﾞｰｽﾄﾛｯｸ手動開要求
      ANI     M389  ; 曲げﾊﾞｯｸﾌﾞｰｽﾄﾛｯｸ開指令
      ANI     M387  ; 曲げﾌﾞｰｽﾄﾛｯｸ開_指令
      ANI     M6009  ; D63=10 ﾊﾞｯｸﾌﾞｰｽﾄﾛｯｸ開
      ANI     M7068  ; D70=680自動運転完了
      ANI     M7127  ; D70=17 ﾊﾞｯｸﾌﾞｰｽﾄﾛｯｸ開指令
      INV
      AND     M2310  ; ﾊﾞｯｸﾌﾞｰｽﾄﾛｯｸ開IL
      ANI     M1  ; 一時停止中
      OR      B1C7  ; SV57ﾌﾞｰｽﾀｰﾛｯｸ 開
      ANB
      ANI     Y1403  ; SV56 ﾌﾞｰｽﾀｰﾛｯｸ 閉
      OUT     Y1404  ; SV57 ﾌﾞｰｽﾀｰﾛｯｸ 開
; ﾊﾞｯｸﾌﾞｰｽﾀ圧抜き
640   LD      SM400  ; 常時 ON
      MPS
      LDI     M2205  ; ﾊﾞｯｸﾌﾞｰｽﾀｰ手動前進要求
      ANI     M2215  ; ﾊﾞｯｸﾌﾞｰｽﾀｰ手動後退要求
      ANI     M2305  ; ﾊﾞｯｸﾌﾞｰｽﾄﾛｯｸ手動閉要求
      ANI     M381  ; 曲げﾊﾞｯｸﾌﾞｰｽﾀ前進_指令
      ANI     M388  ; 曲げﾊﾞｯｸﾌﾞｰｽﾀﾊｰﾌ後退_指令
      ANI     M393  ; 曲げﾊﾞｯｸﾌﾞｰｽﾀﾊｰﾌ前進指令
      ANI     M395  ; 曲げﾊﾞｯｸﾌﾞｰｽﾀﾊｰﾌ前進指令
      INV
      LDI     M380  ; 曲げﾊﾞｯｸﾌﾞｰｽﾄﾛｯｸ閉_指令
      ANI     M6011  ; D63=30 ﾊﾞｯｸﾌﾞｰｽﾀﾊｰﾌ前進
      ANI     M6009  ; D63=10 ﾊﾞｯｸﾌﾞｰｽﾄﾛｯｸ開
      ANI     M6010  ; D63=20 ﾊﾞｯｸﾌﾞｰｽﾀ後退
      ANI     M390  ; 曲げﾊﾞｯｸﾌﾞｰｽﾀ後退指令
      ANI     M391  ; 曲げﾊﾞｯｸﾌﾞｰｽﾄﾛｯｸ閉指令
      INV
      ORB
      ANI     M1  ; 一時停止中
      OR      B1CE  ; SV75ﾊﾞｯｸﾌﾞｰｽﾀｰ 前進側圧抜き
      ANB
      OUT     Y1405  ; SV75 ﾊﾞｯｸﾌﾞｰｽﾀｰ 前進側圧抜き
      MPP
      LDI     M2205  ; ﾊﾞｯｸﾌﾞｰｽﾀｰ手動前進要求
      ANI     M2215  ; ﾊﾞｯｸﾌﾞｰｽﾀｰ手動後退要求
      ANI     M2305  ; ﾊﾞｯｸﾌﾞｰｽﾄﾛｯｸ手動閉要求
      ANI     M381  ; 曲げﾊﾞｯｸﾌﾞｰｽﾀ前進_指令
      ANI     M388  ; 曲げﾊﾞｯｸﾌﾞｰｽﾀﾊｰﾌ後退_指令
      ANI     M393  ; 曲げﾊﾞｯｸﾌﾞｰｽﾀﾊｰﾌ前進指令
      ANI     M395  ; 曲げﾊﾞｯｸﾌﾞｰｽﾀﾊｰﾌ前進指令
      INV
      LDI     M380  ; 曲げﾊﾞｯｸﾌﾞｰｽﾄﾛｯｸ閉_指令
      ANI     M6011  ; D63=30 ﾊﾞｯｸﾌﾞｰｽﾀﾊｰﾌ前進
      ANI     M6009  ; D63=10 ﾊﾞｯｸﾌﾞｰｽﾄﾛｯｸ開
      ANI     M6010  ; D63=20 ﾊﾞｯｸﾌﾞｰｽﾀ後退
      ANI     M390  ; 曲げﾊﾞｯｸﾌﾞｰｽﾀ後退指令
      ANI     M391  ; 曲げﾊﾞｯｸﾌﾞｰｽﾄﾛｯｸ閉指令
      INV
      ORB
      ANI     M1  ; 一時停止中
      OR      B1CF  ; SV76ﾊﾞｯｸﾌﾞｰｽﾀｰ 後退側圧抜き
      ANB
      OUT     Y1406  ; SV76 ﾊﾞｯｸﾌﾞｰｽﾀｰ 後退側圧抜き
; ﾍｯﾄﾞｼﾌﾄ
689   LDI     M2105  ; ﾍﾞﾝﾄﾞﾍｯﾄﾞｼﾌﾄ手動Ｒ大動作要求
      ANI     M2121  ; ﾍﾞﾝﾄﾞﾍｯﾄﾞｼﾌﾄR大移動
      ANI     M6020  ; D60=110 ﾍｯﾄﾞｼﾌﾄ原点復帰
      INV
      AND     M2100  ; ﾍﾞﾝﾄﾞﾍｯﾄﾞｼﾌﾄＲ大IL
      ANI     M1  ; 一時停止中
      OR      B1C5  ; SV55ﾍﾞﾝﾄﾞﾍｯﾄﾞｼﾌﾄ 左移動
      ANI     Y10CC  ; SV54 ﾍﾞﾝﾄﾞﾍｯﾄﾞｼﾌﾄ 右移動
      OUT     Y10CD  ; SV55 ﾍﾞﾝﾄﾞﾍｯﾄﾞｼﾌﾄ 左移動
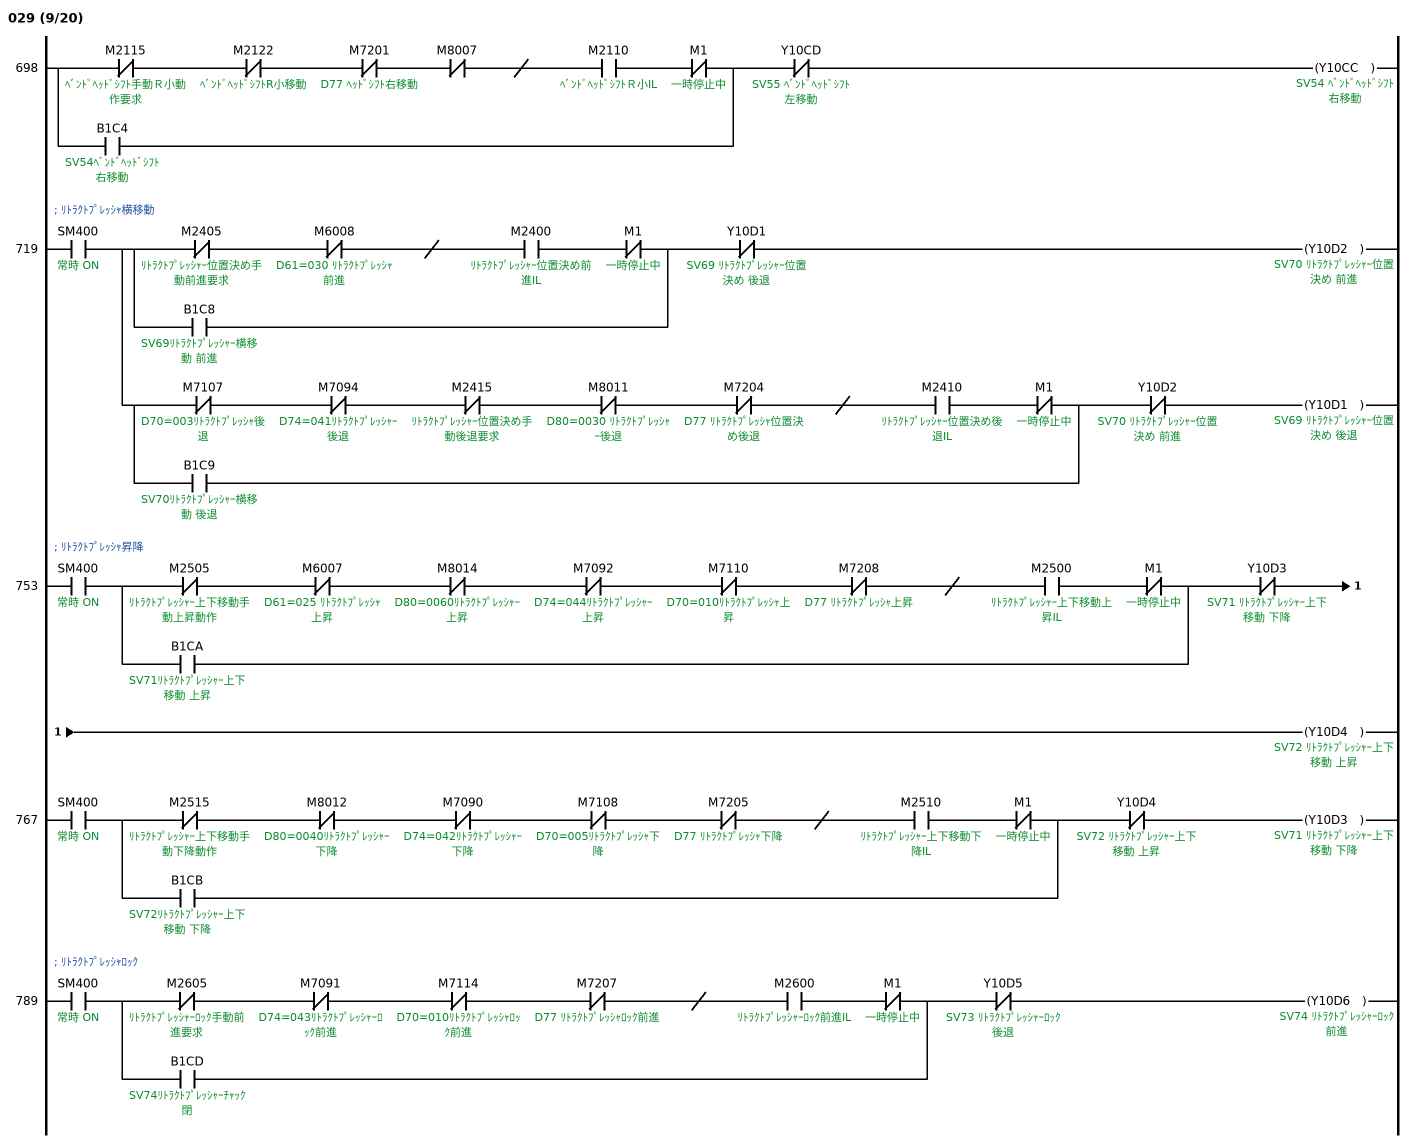
698   LDI     M2115  ; ﾍﾞﾝﾄﾞﾍｯﾄﾞｼﾌﾄ手動Ｒ小動作要求
      ANI     M2122  ; ﾍﾞﾝﾄﾞﾍｯﾄﾞｼﾌﾄR小移動
      ANI     M7201  ; D77 ﾍｯﾄﾞｼﾌﾄ右移動
      ANI     M8007
      INV
      AND     M2110  ; ﾍﾞﾝﾄﾞﾍｯﾄﾞｼﾌﾄＲ小IL
      ANI     M1  ; 一時停止中
      OR      B1C4  ; SV54ﾍﾞﾝﾄﾞﾍｯﾄﾞｼﾌﾄ 右移動
      ANI     Y10CD  ; SV55 ﾍﾞﾝﾄﾞﾍｯﾄﾞｼﾌﾄ 左移動
      OUT     Y10CC  ; SV54 ﾍﾞﾝﾄﾞﾍｯﾄﾞｼﾌﾄ 右移動
; ﾘﾄﾗｸﾄﾌﾟﾚｯｼｬ横移動
719   LD      SM400  ; 常時 ON
      MPS
      LDI     M2405  ; ﾘﾄﾗｸﾄﾌﾟﾚｯｼｬｰ位置決め手動前進要求
      ANI     M6008  ; D61=030 ﾘﾄﾗｸﾄﾌﾟﾚｯｼｬ前進
      INV
      AND     M2400  ; ﾘﾄﾗｸﾄﾌﾟﾚｯｼｬｰ位置決め前進IL
      ANI     M1  ; 一時停止中
      OR      B1C8  ; SV69ﾘﾄﾗｸﾄﾌﾟﾚｯｼｬｰ横移動 前進
      ANB
      ANI     Y10D1  ; SV69 ﾘﾄﾗｸﾄﾌﾟﾚｯｼｬｰ位置決め 後退
      OUT     Y10D2  ; SV70 ﾘﾄﾗｸﾄﾌﾟﾚｯｼｬｰ位置決め 前進
      MPP
      LDI     M7107  ; D70=003ﾘﾄﾗｸﾄﾌﾟﾚｯｼｬ後退
      ANI     M7094  ; D74=041ﾘﾄﾗｸﾄﾌﾟﾚｯｼｬｰ後退
      ANI     M2415  ; ﾘﾄﾗｸﾄﾌﾟﾚｯｼｬｰ位置決め手動後退要求
      ANI     M8011  ; D80=0030 ﾘﾄﾗｸﾄﾌﾟﾚｯｼｬｰ後退
      ANI     M7204  ; D77 ﾘﾄﾗｸﾄﾌﾟﾚｯｼｬ位置決め後退
      INV
      AND     M2410  ; ﾘﾄﾗｸﾄﾌﾟﾚｯｼｬｰ位置決め後退IL
      ANI     M1  ; 一時停止中
      OR      B1C9  ; SV70ﾘﾄﾗｸﾄﾌﾟﾚｯｼｬｰ横移動 後退
      ANB
      ANI     Y10D2  ; SV70 ﾘﾄﾗｸﾄﾌﾟﾚｯｼｬｰ位置決め 前進
      OUT     Y10D1  ; SV69 ﾘﾄﾗｸﾄﾌﾟﾚｯｼｬｰ位置決め 後退
; ﾘﾄﾗｸﾄﾌﾟﾚｯｼｬ昇降
753   LD      SM400  ; 常時 ON
      LDI     M2505  ; ﾘﾄﾗｸﾄﾌﾟﾚｯｼｬｰ上下移動手動上昇動作
      ANI     M6007  ; D61=025 ﾘﾄﾗｸﾄﾌﾟﾚｯｼｬ上昇
      ANI     M8014  ; D80=0060ﾘﾄﾗｸﾄﾌﾟﾚｯｼｬｰ上昇
      ANI     M7092  ; D74=044ﾘﾄﾗｸﾄﾌﾟﾚｯｼｬｰ上昇
      ANI     M7110  ; D70=010ﾘﾄﾗｸﾄﾌﾟﾚｯｼｬ上昇
      ANI     M7208  ; D77 ﾘﾄﾗｸﾄﾌﾟﾚｯｼｬ上昇
      INV
      AND     M2500  ; ﾘﾄﾗｸﾄﾌﾟﾚｯｼｬｰ上下移動上昇IL
      ANI     M1  ; 一時停止中
      OR      B1CA  ; SV71ﾘﾄﾗｸﾄﾌﾟﾚｯｼｬｰ上下移動 上昇
      ANB
      ANI     Y10D3  ; SV71 ﾘﾄﾗｸﾄﾌﾟﾚｯｼｬｰ上下移動 下降
      OUT     Y10D4  ; SV72 ﾘﾄﾗｸﾄﾌﾟﾚｯｼｬｰ上下移動 上昇
767   LD      SM400  ; 常時 ON
      LDI     M2515  ; ﾘﾄﾗｸﾄﾌﾟﾚｯｼｬｰ上下移動手動下降動作
      ANI     M8012  ; D80=0040ﾘﾄﾗｸﾄﾌﾟﾚｯｼｬｰ下降
      ANI     M7090  ; D74=042ﾘﾄﾗｸﾄﾌﾟﾚｯｼｬｰ下降
      ANI     M7108  ; D70=005ﾘﾄﾗｸﾄﾌﾟﾚｯｼｬ下降
      ANI     M7205  ; D77 ﾘﾄﾗｸﾄﾌﾟﾚｯｼｬ下降
      INV
      AND     M2510  ; ﾘﾄﾗｸﾄﾌﾟﾚｯｼｬｰ上下移動下降IL
      ANI     M1  ; 一時停止中
      OR      B1CB  ; SV72ﾘﾄﾗｸﾄﾌﾟﾚｯｼｬｰ上下移動 下降
      ANB
      ANI     Y10D4  ; SV72 ﾘﾄﾗｸﾄﾌﾟﾚｯｼｬｰ上下移動 上昇
      OUT     Y10D3  ; SV71 ﾘﾄﾗｸﾄﾌﾟﾚｯｼｬｰ上下移動 下降
; ﾘﾄﾗｸﾄﾌﾟﾚｯｼｬﾛｯｸ
789   LD      SM400  ; 常時 ON
      LDI     M2605  ; ﾘﾄﾗｸﾄﾌﾟﾚｯｼｬｰﾛｯｸ手動前進要求
      ANI     M7091  ; D74=043ﾘﾄﾗｸﾄﾌﾟﾚｯｼｬｰﾛｯｸ前進
      ANI     M7114  ; D70=010ﾘﾄﾗｸﾄﾌﾟﾚｯｼｬﾛｯｸ前進
      ANI     M7207  ; D77 ﾘﾄﾗｸﾄﾌﾟﾚｯｼｬﾛｯｸ前進
      INV
      AND     M2600  ; ﾘﾄﾗｸﾄﾌﾟﾚｯｼｬｰﾛｯｸ前進IL
      ANI     M1  ; 一時停止中
      OR      B1CD  ; SV74ﾘﾄﾗｸﾄﾌﾟﾚｯｼｬｰﾁｬｯｸ 閉
      ANB
      ANI     Y10D5  ; SV73 ﾘﾄﾗｸﾄﾌﾟﾚｯｼｬｰﾛｯｸ 後退
      OUT     Y10D6  ; SV74 ﾘﾄﾗｸﾄﾌﾟﾚｯｼｬｰﾛｯｸ 前進
